Yaskawa INFORM job: DEMO_ROOF_UPPER_0625_3PAINT_43.JBI

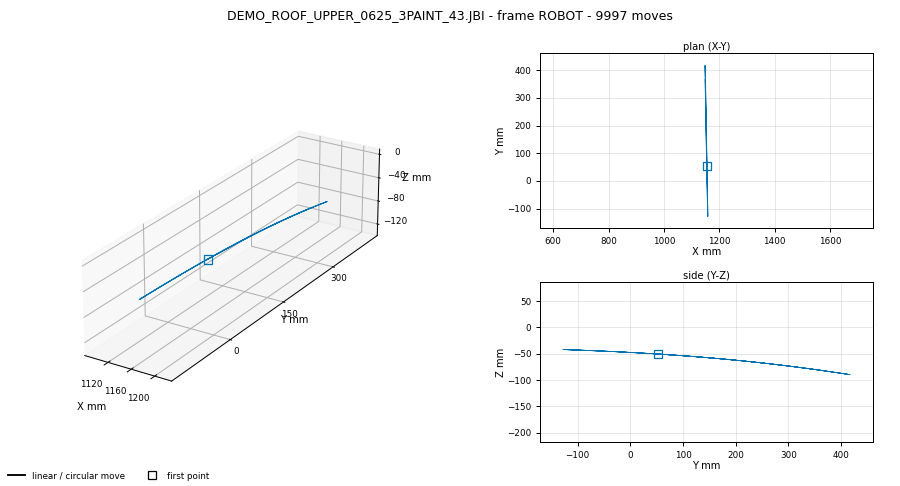
[picture p0: tool path of DEMO_ROOF_UPPER_0625_3PAINT_43.JBI in frame ROBOT, 9997 of 9997 moves have a stored position in this frame; points joined in program order, loops and branches not executed]
/JOB
//NAME DEMO_ROOF_UPPER_0625_3PAINT43
//POS
///NPOS 9997,0,0,0,0,0
///TOOL 0
///USER 0
///POSTYPE ROBOT
///RECTAN
///RCONF 1,0,0,0,0,0,0,0,0,0,0,0,0,0,0,0,0,0,0,0,0,0,0,0
C00000=1156.150,53.320,-50.344,-179.654,6.262,149.031
C00001=1156.144,53.589,-50.362,-179.651,6.263,149.031
C00002=1156.139,53.857,-50.379,-179.648,6.265,149.030
C00003=1156.133,54.126,-50.396,-179.646,6.265,149.030
C00004=1156.128,54.395,-50.413,-179.642,6.267,149.029
C00005=1156.123,54.644,-50.429,-179.640,6.268,149.028
C00006=1156.118,54.893,-50.445,-179.637,6.269,149.028
C00007=1156.113,55.143,-50.461,-179.635,6.270,149.027
C00008=1156.108,55.392,-50.476,-179.632,6.271,149.027
C00009=1156.103,55.641,-50.492,-179.629,6.272,149.026
C00010=1156.098,55.891,-50.508,-179.627,6.274,149.026
C00011=1156.093,56.141,-50.524,-179.624,6.274,149.025
C00012=1156.089,56.390,-50.540,-179.622,6.275,149.025
C00013=1156.083,56.639,-50.556,-179.619,6.277,149.024
C00014=1156.078,56.888,-50.572,-179.617,6.277,149.024
C00015=1156.073,57.138,-50.588,-179.614,6.279,149.023
C00016=1156.068,57.388,-50.604,-179.611,6.279,149.022
C00017=1156.063,57.637,-50.620,-179.608,6.281,149.022
C00018=1156.058,57.887,-50.636,-179.606,6.282,149.022
C00019=1156.054,58.136,-50.653,-179.603,6.283,149.021
C00020=1156.048,58.385,-50.668,-179.601,6.284,149.020
C00021=1156.044,58.635,-50.685,-179.598,6.285,149.020
C00022=1156.038,58.884,-50.700,-179.595,6.286,149.019
C00023=1156.033,59.133,-50.717,-179.592,6.287,149.019
C00024=1156.028,59.383,-50.733,-179.590,6.288,149.018
C00025=1156.023,59.632,-50.749,-179.587,6.290,149.018
C00026=1156.019,59.882,-50.765,-179.585,6.290,149.017
C00027=1156.013,60.131,-50.781,-179.582,6.292,149.017
C00028=1156.009,60.381,-50.797,-179.579,6.293,149.016
C00029=1156.004,60.630,-50.814,-179.577,6.294,149.016
C00030=1155.998,60.880,-50.830,-179.574,6.295,149.015
C00031=1155.993,61.129,-50.846,-179.571,6.296,149.015
C00032=1155.988,61.379,-50.862,-179.569,6.297,149.014
C00033=1155.983,61.628,-50.879,-179.566,6.298,149.013
C00034=1155.979,61.877,-50.895,-179.564,6.299,149.013
C00035=1155.973,62.127,-50.911,-179.561,6.301,149.013
C00036=1155.969,62.376,-50.928,-179.558,6.302,149.012
C00037=1155.963,62.626,-50.943,-179.556,6.303,149.011
C00038=1155.959,62.875,-50.960,-179.553,6.304,149.011
C00039=1155.954,63.124,-50.976,-179.550,6.305,149.010
C00040=1155.948,63.374,-50.993,-179.548,6.306,149.010
C00041=1155.944,63.624,-51.009,-179.545,6.307,149.009
C00042=1155.939,63.873,-51.026,-179.543,6.308,149.009
C00043=1155.934,64.123,-51.042,-179.539,6.310,149.008
C00044=1155.929,64.371,-51.058,-179.537,6.311,149.008
C00045=1155.924,64.621,-51.075,-179.535,6.312,149.007
C00046=1155.919,64.870,-51.092,-179.532,6.313,149.007
C00047=1155.914,65.120,-51.107,-179.529,6.314,149.006
C00048=1155.909,65.369,-51.124,-179.527,6.315,149.006
C00049=1155.904,65.618,-51.140,-179.524,6.317,149.005
C00050=1155.899,65.869,-51.156,-179.521,6.318,149.005
C00051=1155.894,66.118,-51.173,-179.518,6.319,149.004
C00052=1155.889,66.367,-51.190,-179.516,6.320,149.004
C00053=1155.884,66.616,-51.206,-179.514,6.321,149.003
C00054=1155.880,66.865,-51.223,-179.510,6.323,149.003
C00055=1155.875,67.115,-51.239,-179.508,6.323,149.002
C00056=1155.869,67.365,-51.256,-179.505,6.325,149.001
C00057=1155.864,67.614,-51.272,-179.503,6.326,149.001
C00058=1155.859,67.863,-51.289,-179.500,6.327,149.001
C00059=1155.855,68.112,-51.305,-179.497,6.328,149.000
C00060=1155.850,68.362,-51.323,-179.495,6.329,148.999
C00061=1155.844,68.612,-51.338,-179.492,6.330,148.999
C00062=1155.840,68.861,-51.355,-179.489,6.332,148.998
C00063=1155.835,69.111,-51.372,-179.487,6.333,148.998
C00064=1155.830,69.360,-51.389,-179.484,6.334,148.997
C00065=1155.825,69.609,-51.405,-179.481,6.335,148.997
C00066=1155.821,69.859,-51.422,-179.479,6.336,148.996
C00067=1155.815,70.108,-51.439,-179.476,6.338,148.996
C00068=1155.810,70.357,-51.455,-179.474,6.338,148.995
C00069=1155.806,70.607,-51.472,-179.470,6.340,148.995
C00070=1155.800,70.856,-51.489,-179.468,6.341,148.994
C00071=1155.796,71.105,-51.506,-179.466,6.342,148.994
C00072=1155.790,71.356,-51.522,-179.462,6.344,148.993
C00073=1155.785,71.604,-51.539,-179.460,6.344,148.993
C00074=1155.780,71.854,-51.555,-179.457,6.346,148.992
C00075=1155.775,72.104,-51.572,-179.455,6.347,148.992
C00076=1155.770,72.352,-51.589,-179.452,6.348,148.991
C00077=1155.766,72.602,-51.605,-179.449,6.350,148.991
C00078=1155.761,72.851,-51.623,-179.447,6.350,148.990
C00079=1155.756,73.100,-51.640,-179.444,6.352,148.990
C00080=1155.750,73.350,-51.657,-179.441,6.353,148.989
C00081=1155.746,73.599,-51.674,-179.439,6.354,148.989
C00082=1155.741,73.849,-51.690,-179.436,6.355,148.988
C00083=1155.736,74.098,-51.707,-179.433,6.357,148.987
C00084=1155.731,74.347,-51.724,-179.430,6.358,148.987
C00085=1155.726,74.597,-51.741,-179.428,6.359,148.987
C00086=1155.721,74.847,-51.758,-179.425,6.360,148.986
C00087=1155.716,75.096,-51.775,-179.423,6.361,148.986
C00088=1155.711,75.345,-51.791,-179.420,6.363,148.985
C00089=1155.706,75.595,-51.809,-179.417,6.364,148.984
C00090=1155.702,75.844,-51.826,-179.415,6.365,148.984
C00091=1155.696,76.093,-51.843,-179.412,6.367,148.984
C00092=1155.691,76.342,-51.860,-179.409,6.367,148.983
C00093=1155.686,76.592,-51.877,-179.407,6.369,148.983
C00094=1155.682,76.842,-51.894,-179.404,6.371,148.982
C00095=1155.676,77.091,-51.910,-179.401,6.371,148.981
C00096=1155.672,77.340,-51.928,-179.399,6.373,148.981
C00097=1155.667,77.589,-51.945,-179.396,6.373,148.980
C00098=1155.662,77.839,-51.962,-179.393,6.375,148.980
C00099=1155.657,78.089,-51.979,-179.391,6.377,148.979
C00100=1155.652,78.337,-51.996,-179.388,6.377,148.979
C00101=1155.647,78.587,-52.013,-179.385,6.379,148.978
C00102=1155.642,78.836,-52.030,-179.382,6.381,148.978
C00103=1155.637,79.086,-52.047,-179.380,6.381,148.977
C00104=1155.632,79.335,-52.065,-179.377,6.383,148.977
C00105=1155.627,79.603,-52.083,-179.374,6.384,148.976
C00106=1155.622,79.872,-52.102,-179.372,6.385,148.976
C00107=1155.616,80.141,-52.120,-179.369,6.387,148.975
C00108=1155.611,80.409,-52.138,-179.366,6.388,148.975
C00109=1155.606,80.658,-52.156,-179.363,6.390,148.974
C00110=1155.602,80.907,-52.173,-179.360,6.390,148.974
C00111=1155.596,81.157,-52.190,-179.358,6.392,148.973
C00112=1155.591,81.406,-52.208,-179.355,6.393,148.973
C00113=1155.586,81.655,-52.224,-179.352,6.394,148.972
C00114=1155.581,81.904,-52.242,-179.350,6.396,148.972
C00115=1155.576,82.154,-52.259,-179.347,6.397,148.971
C00116=1155.572,82.403,-52.276,-179.344,6.398,148.971
C00117=1155.567,82.653,-52.294,-179.341,6.400,148.970
C00118=1155.562,82.902,-52.311,-179.339,6.401,148.970
C00119=1155.557,83.151,-52.329,-179.336,6.402,148.969
C00120=1155.552,83.401,-52.346,-179.333,6.403,148.969
C00121=1155.547,83.650,-52.364,-179.331,6.404,148.968
C00122=1155.542,83.899,-52.380,-179.329,6.406,148.968
C00123=1155.537,84.148,-52.398,-179.325,6.407,148.967
C00124=1155.532,84.398,-52.416,-179.323,6.408,148.967
C00125=1155.527,84.647,-52.434,-179.320,6.410,148.966
C00126=1155.523,84.897,-52.450,-179.317,6.411,148.966
C00127=1155.518,85.146,-52.468,-179.315,6.412,148.965
C00128=1155.513,85.396,-52.485,-179.312,6.414,148.965
C00129=1155.508,85.645,-52.503,-179.309,6.415,148.964
C00130=1155.503,85.894,-52.520,-179.307,6.416,148.964
C00131=1155.498,86.143,-52.538,-179.304,6.418,148.963
C00132=1155.493,86.393,-52.555,-179.301,6.419,148.963
C00133=1155.488,86.642,-52.573,-179.299,6.420,148.962
C00134=1155.484,86.892,-52.590,-179.296,6.421,148.962
C00135=1155.479,87.141,-52.608,-179.293,6.423,148.961
C00136=1155.474,87.390,-52.626,-179.290,6.424,148.961
C00137=1155.469,87.640,-52.643,-179.288,6.425,148.960
C00138=1155.464,87.889,-52.661,-179.285,6.427,148.960
C00139=1155.460,88.138,-52.679,-179.282,6.428,148.959
C00140=1155.454,88.388,-52.696,-179.280,6.429,148.959
C00141=1155.449,88.637,-52.714,-179.277,6.431,148.959
C00142=1155.445,88.886,-52.732,-179.274,6.432,148.958
C00143=1155.439,89.136,-52.749,-179.272,6.433,148.957
C00144=1155.434,89.385,-52.767,-179.269,6.435,148.957
C00145=1155.429,89.634,-52.785,-179.266,6.437,148.957
C00146=1155.425,89.884,-52.802,-179.264,6.437,148.956
C00147=1155.420,90.133,-52.820,-179.261,6.439,148.956
C00148=1155.415,90.382,-52.838,-179.258,6.440,148.955
C00149=1155.410,90.631,-52.856,-179.255,6.442,148.954
C00150=1155.405,90.881,-52.873,-179.253,6.443,148.954
C00151=1155.400,91.130,-52.891,-179.250,6.444,148.954
C00152=1155.395,91.380,-52.909,-179.247,6.446,148.953
C00153=1155.390,91.629,-52.927,-179.245,6.446,148.953
C00154=1155.385,91.878,-52.944,-179.242,6.448,148.952
C00155=1155.380,92.128,-52.962,-179.239,6.450,148.952
C00156=1155.376,92.377,-52.979,-179.236,6.451,148.951
C00157=1155.371,92.626,-52.997,-179.234,6.452,148.951
C00158=1155.366,92.875,-53.015,-179.231,6.454,148.950
C00159=1155.361,93.124,-53.033,-179.229,6.455,148.950
C00160=1155.356,93.374,-53.051,-179.226,6.456,148.949
C00161=1155.351,93.623,-53.069,-179.223,6.458,148.949
C00162=1155.346,93.872,-53.087,-179.221,6.459,148.948
C00163=1155.342,94.122,-53.105,-179.218,6.461,148.948
C00164=1155.337,94.371,-53.123,-179.215,6.462,148.947
C00165=1155.332,94.620,-53.141,-179.212,6.463,148.947
C00166=1155.327,94.870,-53.159,-179.210,6.465,148.946
C00167=1155.322,95.119,-53.177,-179.207,6.466,148.946
C00168=1155.317,95.368,-53.195,-179.204,6.467,148.945
C00169=1155.312,95.617,-53.213,-179.202,6.469,148.945
C00170=1155.308,95.866,-53.231,-179.199,6.471,148.945
C00171=1155.303,96.115,-53.249,-179.196,6.471,148.944
C00172=1155.298,96.366,-53.268,-179.194,6.473,148.943
C00173=1155.292,96.615,-53.285,-179.191,6.474,148.943
C00174=1155.287,96.865,-53.303,-179.188,6.476,148.943
C00175=1155.283,97.113,-53.322,-179.185,6.477,148.942
C00176=1155.278,97.362,-53.340,-179.183,6.478,148.942
C00177=1155.273,97.612,-53.358,-179.180,6.480,148.941
C00178=1155.269,97.861,-53.376,-179.177,6.482,148.941
C00179=1155.264,98.111,-53.394,-179.174,6.483,148.940
C00180=1155.259,98.360,-53.412,-179.172,6.484,148.940
C00181=1155.254,98.609,-53.430,-179.169,6.486,148.939
C00182=1155.249,98.858,-53.448,-179.166,6.487,148.939
C00183=1155.243,99.108,-53.467,-179.163,6.489,148.938
C00184=1155.239,99.357,-53.485,-179.161,6.490,148.938
C00185=1155.234,99.607,-53.503,-179.158,6.491,148.937
C00186=1155.229,99.856,-53.521,-179.156,6.493,148.937
C00187=1155.224,100.105,-53.539,-179.152,6.494,148.936
C00188=1155.220,100.354,-53.557,-179.150,6.495,148.936
C00189=1155.215,100.604,-53.576,-179.148,6.497,148.935
C00190=1155.210,100.853,-53.594,-179.145,6.499,148.935
C00191=1155.205,101.102,-53.612,-179.142,6.500,148.934
C00192=1155.200,101.351,-53.630,-179.139,6.502,148.934
C00193=1155.196,101.601,-53.649,-179.137,6.502,148.934
C00194=1155.190,101.850,-53.668,-179.134,6.504,148.933
C00195=1155.185,102.099,-53.686,-179.131,6.506,148.933
C00196=1155.181,102.348,-53.704,-179.128,6.507,148.932
C00197=1155.176,102.598,-53.722,-179.126,6.508,148.932
C00198=1155.172,102.847,-53.741,-179.123,6.510,148.931
C00199=1155.166,103.096,-53.760,-179.121,6.511,148.931
C00200=1155.161,103.345,-53.778,-179.117,6.513,148.930
C00201=1155.157,103.595,-53.796,-179.115,6.514,148.930
C00202=1155.151,103.844,-53.815,-179.113,6.515,148.929
C00203=1155.146,104.093,-53.833,-179.110,6.517,148.929
C00204=1155.142,104.343,-53.851,-179.107,6.518,148.928
C00205=1155.138,104.592,-53.870,-179.104,6.520,148.928
C00206=1155.132,104.841,-53.889,-179.101,6.522,148.928
C00207=1155.127,105.090,-53.907,-179.099,6.523,148.927
C00208=1155.123,105.340,-53.926,-179.096,6.524,148.927
C00209=1155.117,105.608,-53.946,-179.093,6.526,148.926
C00210=1155.112,105.877,-53.965,-179.090,6.527,148.926
C00211=1155.107,106.145,-53.986,-179.087,6.529,148.925
C00212=1155.102,106.413,-54.006,-179.084,6.530,148.925
C00213=1155.096,106.663,-54.024,-179.082,6.532,148.924
C00214=1155.092,106.912,-54.043,-179.079,6.534,148.924
C00215=1155.088,107.161,-54.061,-179.076,6.536,148.923
C00216=1155.082,107.410,-54.081,-179.073,6.537,148.923
C00217=1155.077,107.659,-54.099,-179.070,6.539,148.922
C00218=1155.073,107.909,-54.118,-179.068,6.539,148.922
C00219=1155.068,108.158,-54.136,-179.065,6.541,148.922
C00220=1155.063,108.407,-54.155,-179.063,6.543,148.921
C00221=1155.058,108.657,-54.174,-179.060,6.544,148.921
C00222=1155.053,108.905,-54.193,-179.057,6.546,148.920
C00223=1155.048,109.155,-54.211,-179.054,6.548,148.920
C00224=1155.044,109.404,-54.230,-179.052,6.548,148.919
C00225=1155.039,109.653,-54.248,-179.049,6.550,148.919
C00226=1155.034,109.903,-54.268,-179.046,6.552,148.918
C00227=1155.029,110.152,-54.286,-179.043,6.553,148.918
C00228=1155.024,110.401,-54.305,-179.041,6.555,148.917
C00229=1155.019,110.651,-54.323,-179.038,6.557,148.917
C00230=1155.014,110.900,-54.343,-179.036,6.558,148.917
C00231=1155.010,111.149,-54.362,-179.033,6.559,148.916
C00232=1155.004,111.398,-54.380,-179.030,6.561,148.916
C00233=1155.000,111.647,-54.399,-179.027,6.562,148.915
C00234=1154.995,111.897,-54.418,-179.024,6.564,148.915
C00235=1154.990,112.146,-54.437,-179.022,6.566,148.914
C00236=1154.985,112.395,-54.456,-179.019,6.567,148.914
C00237=1154.981,112.645,-54.474,-179.016,6.568,148.913
C00238=1154.976,112.894,-54.494,-179.014,6.570,148.913
C00239=1154.971,113.143,-54.513,-179.011,6.571,148.913
C00240=1154.966,113.392,-54.531,-179.008,6.573,148.912
C00241=1154.961,113.642,-54.551,-179.005,6.575,148.912
C00242=1154.956,113.890,-54.570,-179.003,6.576,148.911
C00243=1154.951,114.140,-54.589,-178.999,6.578,148.911
C00244=1154.947,114.389,-54.607,-178.997,6.579,148.910
C00245=1154.942,114.639,-54.627,-178.995,6.580,148.910
C00246=1154.937,114.887,-54.646,-178.992,6.582,148.909
C00247=1154.932,115.137,-54.665,-178.989,6.584,148.909
C00248=1154.927,115.386,-54.684,-178.986,6.585,148.909
C00249=1154.923,115.635,-54.703,-178.983,6.587,148.908
C00250=1154.917,115.884,-54.722,-178.981,6.589,148.908
C00251=1154.913,116.134,-54.742,-178.978,6.590,148.907
C00252=1154.908,116.382,-54.761,-178.975,6.592,148.907
C00253=1154.903,116.632,-54.780,-178.973,6.593,148.906
C00254=1154.898,116.881,-54.798,-178.970,6.595,148.906
C00255=1154.894,117.131,-54.818,-178.968,6.596,148.906
C00256=1154.888,117.380,-54.837,-178.964,6.598,148.905
C00257=1154.884,117.629,-54.857,-178.962,6.599,148.905
C00258=1154.879,117.878,-54.876,-178.959,6.601,148.904
C00259=1154.874,118.127,-54.895,-178.956,6.603,148.904
C00260=1154.870,118.377,-54.915,-178.953,6.604,148.903
C00261=1154.865,118.625,-54.934,-178.951,6.606,148.903
C00262=1154.860,118.875,-54.953,-178.948,6.608,148.903
C00263=1154.855,119.124,-54.972,-178.945,6.608,148.902
C00264=1154.851,119.373,-54.992,-178.943,6.610,148.901
C00265=1154.845,119.623,-55.010,-178.940,6.612,148.901
C00266=1154.840,119.872,-55.030,-178.937,6.613,148.901
C00267=1154.836,120.122,-55.049,-178.935,6.615,148.900
C00268=1154.831,120.370,-55.068,-178.932,6.617,148.900
C00269=1154.826,120.620,-55.088,-178.929,6.619,148.899
C00270=1154.821,120.869,-55.107,-178.926,6.620,148.899
C00271=1154.817,121.118,-55.127,-178.923,6.622,148.898
C00272=1154.812,121.367,-55.147,-178.920,6.623,148.898
C00273=1154.807,121.616,-55.166,-178.918,6.625,148.898
C00274=1154.802,121.865,-55.185,-178.915,6.627,148.897
C00275=1154.797,122.114,-55.205,-178.912,6.629,148.897
C00276=1154.792,122.364,-55.224,-178.910,6.630,148.896
C00277=1154.788,122.613,-55.244,-178.907,6.631,148.896
C00278=1154.783,122.862,-55.263,-178.905,6.633,148.896
C00279=1154.778,123.112,-55.282,-178.902,6.634,148.895
C00280=1154.774,123.361,-55.302,-178.899,6.636,148.895
C00281=1154.768,123.610,-55.321,-178.896,6.638,148.894
C00282=1154.764,123.859,-55.342,-178.893,6.639,148.894
C00283=1154.759,124.108,-55.361,-178.891,6.641,148.893
C00284=1154.754,124.357,-55.380,-178.888,6.643,148.893
C00285=1154.750,124.607,-55.400,-178.885,6.644,148.893
C00286=1154.745,124.856,-55.419,-178.883,6.646,148.892
C00287=1154.740,125.104,-55.439,-178.880,6.648,148.892
C00288=1154.735,125.354,-55.459,-178.877,6.650,148.891
C00289=1154.730,125.604,-55.479,-178.874,6.651,148.891
C00290=1154.725,125.852,-55.498,-178.871,6.653,148.890
C00291=1154.721,126.101,-55.518,-178.868,6.654,148.890
C00292=1154.716,126.351,-55.538,-178.866,6.656,148.890
C00293=1154.711,126.600,-55.557,-178.863,6.658,148.889
C00294=1154.706,126.849,-55.577,-178.860,6.659,148.889
C00295=1154.701,127.098,-55.597,-178.858,6.661,148.888
C00296=1154.697,127.348,-55.616,-178.855,6.663,148.888
C00297=1154.692,127.596,-55.636,-178.852,6.665,148.888
C00298=1154.688,127.845,-55.656,-178.849,6.666,148.887
C00299=1154.683,128.095,-55.676,-178.847,6.667,148.887
C00300=1154.678,128.345,-55.695,-178.844,6.669,148.886
C00301=1154.673,128.593,-55.715,-178.841,6.670,148.886
C00302=1154.668,128.842,-55.735,-178.839,6.672,148.885
C00303=1154.664,129.092,-55.755,-178.836,6.674,148.885
C00304=1154.659,129.341,-55.775,-178.833,6.675,148.885
C00305=1154.654,129.590,-55.794,-178.831,6.677,148.884
C00306=1154.649,129.839,-55.815,-178.828,6.679,148.884
C00307=1154.644,130.089,-55.835,-178.825,6.681,148.883
C00308=1154.639,130.338,-55.855,-178.822,6.682,148.883
C00309=1154.634,130.586,-55.875,-178.820,6.684,148.883
C00310=1154.629,130.836,-55.894,-178.817,6.686,148.882
C00311=1154.625,131.085,-55.915,-178.814,6.687,148.882
C00312=1154.620,131.334,-55.934,-178.812,6.689,148.881
C00313=1154.616,131.602,-55.956,-178.808,6.691,148.881
C00314=1154.610,131.871,-55.978,-178.805,6.693,148.880
C00315=1154.605,132.140,-55.999,-178.802,6.695,148.880
C00316=1154.600,132.408,-56.021,-178.800,6.696,148.880
C00317=1154.595,132.658,-56.041,-178.797,6.698,148.879
C00318=1154.590,132.906,-56.061,-178.794,6.700,148.879
C00319=1154.585,133.156,-56.081,-178.792,6.702,148.879
C00320=1154.581,133.405,-56.101,-178.789,6.703,148.878
C00321=1154.576,133.654,-56.121,-178.786,6.705,148.878
C00322=1154.571,133.904,-56.142,-178.783,6.706,148.877
C00323=1154.566,134.153,-56.162,-178.780,6.708,148.877
C00324=1154.561,134.401,-56.181,-178.778,6.710,148.876
C00325=1154.557,134.650,-56.202,-178.775,6.712,148.876
C00326=1154.552,134.899,-56.222,-178.772,6.714,148.876
C00327=1154.547,135.149,-56.242,-178.769,6.716,148.875
C00328=1154.542,135.398,-56.263,-178.766,6.718,148.875
C00329=1154.538,135.647,-56.283,-178.763,6.719,148.874
C00330=1154.533,135.897,-56.303,-178.761,6.721,148.874
C00331=1154.529,136.146,-56.323,-178.758,6.723,148.874
C00332=1154.523,136.395,-56.344,-178.755,6.724,148.873
C00333=1154.518,136.644,-56.363,-178.753,6.726,148.873
C00334=1154.514,136.893,-56.384,-178.750,6.728,148.872
C00335=1154.509,137.142,-56.404,-178.747,6.730,148.872
C00336=1154.504,137.391,-56.425,-178.744,6.731,148.872
C00337=1154.499,137.640,-56.445,-178.742,6.733,148.871
C00338=1154.495,137.889,-56.465,-178.739,6.735,148.871
C00339=1154.490,138.139,-56.486,-178.736,6.736,148.870
C00340=1154.485,138.388,-56.506,-178.734,6.738,148.870
C00341=1154.481,138.637,-56.527,-178.731,6.740,148.870
C00342=1154.476,138.886,-56.546,-178.728,6.742,148.869
C00343=1154.471,139.135,-56.567,-178.725,6.743,148.869
C00344=1154.466,139.384,-56.588,-178.723,6.745,148.869
C00345=1154.462,139.633,-56.608,-178.720,6.747,148.868
C00346=1154.457,139.883,-56.629,-178.717,6.748,148.868
C00347=1154.452,140.132,-56.649,-178.714,6.751,148.867
C00348=1154.448,140.380,-56.670,-178.711,6.753,148.867
C00349=1154.442,140.630,-56.690,-178.709,6.754,148.867
C00350=1154.438,140.879,-56.710,-178.706,6.756,148.866
C00351=1154.433,141.129,-56.731,-178.703,6.758,148.866
C00352=1154.428,141.377,-56.752,-178.700,6.760,148.865
C00353=1154.424,141.626,-56.772,-178.698,6.761,148.865
C00354=1154.419,141.876,-56.793,-178.695,6.763,148.865
C00355=1154.414,142.125,-56.813,-178.692,6.765,148.864
C00356=1154.409,142.374,-56.834,-178.690,6.767,148.864
C00357=1154.405,142.623,-56.855,-178.687,6.768,148.864
C00358=1154.400,142.872,-56.875,-178.684,6.770,148.863
C00359=1154.395,143.121,-56.896,-178.682,6.772,148.863
C00360=1154.391,143.370,-56.917,-178.678,6.774,148.862
C00361=1154.386,143.619,-56.938,-178.676,6.776,148.862
C00362=1154.381,143.868,-56.958,-178.673,6.778,148.862
C00363=1154.376,144.117,-56.979,-178.670,6.779,148.861
C00364=1154.371,144.366,-56.999,-178.667,6.781,148.861
C00365=1154.366,144.616,-57.020,-178.665,6.783,148.860
C00366=1154.362,144.864,-57.041,-178.662,6.785,148.860
C00367=1154.357,145.113,-57.062,-178.659,6.786,148.860
C00368=1154.353,145.362,-57.083,-178.657,6.788,148.859
C00369=1154.347,145.611,-57.104,-178.654,6.790,148.859
C00370=1154.343,145.860,-57.124,-178.651,6.792,148.859
C00371=1154.338,146.110,-57.145,-178.648,6.794,148.858
C00372=1154.334,146.359,-57.166,-178.645,6.796,148.858
C00373=1154.329,146.608,-57.187,-178.643,6.798,148.858
C00374=1154.325,146.857,-57.208,-178.640,6.800,148.857
C00375=1154.319,147.106,-57.229,-178.638,6.801,148.857
C00376=1154.315,147.355,-57.249,-178.635,6.803,148.856
C00377=1154.310,147.604,-57.270,-178.632,6.805,148.856
C00378=1154.305,147.853,-57.292,-178.629,6.806,148.856
C00379=1154.301,148.102,-57.312,-178.626,6.809,148.855
C00380=1154.296,148.352,-57.333,-178.623,6.811,148.855
C00381=1154.292,148.601,-57.354,-178.621,6.812,148.855
C00382=1154.287,148.850,-57.375,-178.618,6.814,148.854
C00383=1154.281,149.099,-57.396,-178.615,6.816,148.854
C00384=1154.277,149.348,-57.417,-178.613,6.818,148.853
C00385=1154.272,149.597,-57.438,-178.610,6.819,148.853
C00386=1154.267,149.846,-57.459,-178.607,6.822,148.853
C00387=1154.263,150.095,-57.480,-178.604,6.824,148.852
C00388=1154.258,150.345,-57.501,-178.601,6.825,148.852
C00389=1154.253,150.593,-57.523,-178.598,6.827,148.851
C00390=1154.249,150.842,-57.543,-178.596,6.829,148.851
C00391=1154.244,151.091,-57.565,-178.594,6.831,148.851
C00392=1154.239,151.341,-57.586,-178.591,6.833,148.851
C00393=1154.235,151.590,-57.607,-178.588,6.835,148.850
C00394=1154.230,151.838,-57.628,-178.585,6.837,148.850
C00395=1154.225,152.088,-57.649,-178.582,6.839,148.849
C00396=1154.220,152.336,-57.671,-178.579,6.840,148.849
C00397=1154.216,152.586,-57.692,-178.577,6.842,148.849
C00398=1154.211,152.835,-57.713,-178.574,6.844,148.848
C00399=1154.206,153.084,-57.734,-178.571,6.846,148.848
C00400=1154.201,153.333,-57.755,-178.568,6.848,148.848
C00401=1154.197,153.581,-57.776,-178.566,6.850,148.847
C00402=1154.192,153.831,-57.798,-178.563,6.852,148.847
C00403=1154.187,154.080,-57.819,-178.560,6.854,148.847
C00404=1154.182,154.329,-57.840,-178.558,6.855,148.846
C00405=1154.177,154.578,-57.862,-178.554,6.858,148.846
C00406=1154.174,154.827,-57.883,-178.552,6.860,148.846
C00407=1154.168,155.076,-57.904,-178.549,6.861,148.845
C00408=1154.164,155.325,-57.926,-178.546,6.863,148.845
C00409=1154.159,155.575,-57.947,-178.544,6.865,148.844
C00410=1154.154,155.823,-57.969,-178.541,6.867,148.844
C00411=1154.149,156.073,-57.990,-178.538,6.869,148.844
C00412=1154.145,156.321,-58.011,-178.535,6.871,148.843
C00413=1154.141,156.570,-58.033,-178.533,6.873,148.843
C00414=1154.135,156.820,-58.054,-178.530,6.875,148.843
C00415=1154.131,157.068,-58.076,-178.527,6.876,148.842
C00416=1154.126,157.318,-58.098,-178.524,6.879,148.842
C00417=1154.122,157.587,-58.121,-178.521,6.881,148.842
C00418=1154.115,157.855,-58.144,-178.518,6.883,148.841
C00419=1154.111,158.124,-58.167,-178.515,6.885,148.841
C00420=1154.106,158.393,-58.191,-178.513,6.887,148.841
C00421=1154.101,158.642,-58.213,-178.509,6.889,148.840
C00422=1154.096,158.892,-58.234,-178.507,6.891,148.840
C00423=1154.091,159.140,-58.255,-178.504,6.893,148.839
C00424=1154.087,159.390,-58.277,-178.502,6.895,148.839
C00425=1154.082,159.638,-58.299,-178.499,6.896,148.839
C00426=1154.077,159.888,-58.320,-178.496,6.899,148.839
C00427=1154.073,160.137,-58.342,-178.493,6.901,148.838
C00428=1154.068,160.386,-58.364,-178.490,6.902,148.838
C00429=1154.064,160.635,-58.386,-178.488,6.904,148.837
C00430=1154.059,160.884,-58.407,-178.484,6.907,148.837
C00431=1154.053,161.133,-58.428,-178.482,6.909,148.837
C00432=1154.049,161.382,-58.450,-178.479,6.911,148.836
C00433=1154.044,161.631,-58.472,-178.477,6.912,148.836
C00434=1154.040,161.880,-58.494,-178.474,6.914,148.836
C00435=1154.035,162.129,-58.516,-178.471,6.917,148.835
C00436=1154.030,162.377,-58.538,-178.468,6.918,148.835
C00437=1154.026,162.627,-58.560,-178.466,6.920,148.835
C00438=1154.021,162.875,-58.581,-178.463,6.922,148.834
C00439=1154.017,163.125,-58.603,-178.460,6.925,148.834
C00440=1154.012,163.373,-58.625,-178.457,6.926,148.834
C00441=1154.008,163.623,-58.647,-178.454,6.928,148.833
C00442=1154.003,163.871,-58.669,-178.452,6.930,148.833
C00443=1153.998,164.120,-58.690,-178.449,6.933,148.833
C00444=1153.994,164.369,-58.712,-178.446,6.935,148.832
C00445=1153.989,164.618,-58.734,-178.444,6.936,148.832
C00446=1153.985,164.867,-58.756,-178.441,6.938,148.832
C00447=1153.979,165.116,-58.778,-178.438,6.941,148.831
C00448=1153.975,165.366,-58.800,-178.435,6.943,148.831
C00449=1153.970,165.614,-58.822,-178.433,6.944,148.831
C00450=1153.966,165.864,-58.844,-178.430,6.946,148.831
C00451=1153.961,166.112,-58.866,-178.427,6.949,148.830
C00452=1153.956,166.362,-58.888,-178.424,6.950,148.830
C00453=1153.952,166.610,-58.910,-178.421,6.952,148.829
C00454=1153.947,166.860,-58.932,-178.419,6.954,148.829
C00455=1153.942,167.108,-58.954,-178.416,6.957,148.829
C00456=1153.937,167.358,-58.976,-178.413,6.959,148.829
C00457=1153.933,167.606,-58.998,-178.410,6.960,148.828
C00458=1153.929,167.855,-59.020,-178.407,6.963,148.828
C00459=1153.923,168.104,-59.043,-178.405,6.965,148.828
C00460=1153.919,168.353,-59.065,-178.402,6.967,148.827
C00461=1153.914,168.602,-59.086,-178.399,6.968,148.827
C00462=1153.910,168.851,-59.109,-178.396,6.971,148.827
C00463=1153.905,169.100,-59.132,-178.394,6.973,148.826
C00464=1153.900,169.349,-59.154,-178.391,6.975,148.826
C00465=1153.896,169.598,-59.176,-178.388,6.977,148.826
C00466=1153.890,169.847,-59.198,-178.385,6.979,148.825
C00467=1153.886,170.096,-59.221,-178.383,6.981,148.825
C00468=1153.881,170.345,-59.242,-178.380,6.983,148.825
C00469=1153.877,170.594,-59.264,-178.377,6.985,148.824
C00470=1153.871,170.843,-59.287,-178.374,6.987,148.824
C00471=1153.868,171.092,-59.309,-178.372,6.989,148.824
C00472=1153.863,171.341,-59.331,-178.369,6.992,148.824
C00473=1153.858,171.590,-59.354,-178.366,6.994,148.823
C00474=1153.854,171.839,-59.376,-178.364,6.995,148.823
C00475=1153.849,172.087,-59.398,-178.360,6.998,148.823
C00476=1153.844,172.336,-59.422,-178.358,7.000,148.822
C00477=1153.840,172.586,-59.444,-178.355,7.002,148.822
C00478=1153.834,172.835,-59.466,-178.353,7.003,148.822
C00479=1153.830,173.083,-59.489,-178.349,7.006,148.821
C00480=1153.826,173.333,-59.511,-178.347,7.008,148.821
C00481=1153.821,173.581,-59.534,-178.344,7.010,148.821
C00482=1153.816,173.831,-59.556,-178.341,7.012,148.820
C00483=1153.811,174.080,-59.578,-178.338,7.014,148.820
C00484=1153.807,174.328,-59.601,-178.336,7.016,148.820
C00485=1153.803,174.578,-59.623,-178.333,7.019,148.820
C00486=1153.798,174.827,-59.646,-178.330,7.020,148.819
C00487=1153.793,175.075,-59.668,-178.328,7.022,148.819
C00488=1153.788,175.324,-59.691,-178.325,7.025,148.819
C00489=1153.784,175.574,-59.713,-178.322,7.027,148.818
C00490=1153.779,175.822,-59.736,-178.319,7.029,148.818
C00491=1153.775,176.071,-59.759,-178.316,7.031,148.818
C00492=1153.770,176.320,-59.782,-178.314,7.033,148.817
C00493=1153.765,176.568,-59.804,-178.311,7.035,148.817
C00494=1153.760,176.818,-59.827,-178.308,7.038,148.817
C00495=1153.756,177.067,-59.849,-178.305,7.039,148.816
C00496=1153.751,177.316,-59.872,-178.303,7.041,148.816
C00497=1153.747,177.564,-59.894,-178.300,7.044,148.816
C00498=1153.742,177.813,-59.918,-178.297,7.046,148.816
C00499=1153.738,178.063,-59.940,-178.295,7.048,148.815
C00500=1153.732,178.311,-59.963,-178.292,7.050,148.815
C00501=1153.728,178.560,-59.986,-178.289,7.052,148.815
C00502=1153.723,178.809,-60.008,-178.286,7.055,148.814
C00503=1153.720,179.058,-60.031,-178.283,7.057,148.814
C00504=1153.714,179.306,-60.054,-178.281,7.059,148.814
C00505=1153.710,179.555,-60.077,-178.277,7.061,148.814
C00506=1153.705,179.805,-60.099,-178.275,7.063,148.813
C00507=1153.701,180.054,-60.123,-178.272,7.065,148.813
C00508=1153.697,180.303,-60.146,-178.269,7.067,148.813
C00509=1153.691,180.551,-60.169,-178.267,7.070,148.813
C00510=1153.686,180.801,-60.191,-178.264,7.071,148.812
C00511=1153.682,181.049,-60.214,-178.261,7.074,148.812
C00512=1153.678,181.298,-60.237,-178.259,7.076,148.812
C00513=1153.672,181.547,-60.260,-178.256,7.079,148.811
C00514=1153.668,181.795,-60.283,-178.253,7.080,148.811
C00515=1153.663,182.045,-60.306,-178.251,7.082,148.811
C00516=1153.659,182.294,-60.329,-178.247,7.085,148.810
C00517=1153.655,182.543,-60.352,-178.245,7.087,148.810
C00518=1153.650,182.792,-60.375,-178.241,7.089,148.810
C00519=1153.645,183.040,-60.398,-178.239,7.091,148.810
C00520=1153.641,183.289,-60.421,-178.237,7.093,148.809
C00521=1153.635,183.559,-60.446,-178.233,7.096,148.809
C00522=1153.630,183.828,-60.471,-178.230,7.099,148.809
C00523=1153.626,184.099,-60.496,-178.228,7.100,148.808
C00524=1153.621,184.368,-60.521,-178.224,7.103,148.808
C00525=1153.615,184.617,-60.544,-178.222,7.105,148.808
C00526=1153.611,184.866,-60.567,-178.219,7.108,148.808
C00527=1153.607,185.114,-60.590,-178.216,7.109,148.807
C00528=1153.602,185.363,-60.613,-178.213,7.112,148.807
C00529=1153.597,185.612,-60.637,-178.211,7.114,148.807
C00530=1153.593,185.862,-60.660,-178.208,7.116,148.806
C00531=1153.588,186.111,-60.683,-178.205,7.118,148.806
C00532=1153.584,186.359,-60.707,-178.203,7.120,148.806
C00533=1153.580,186.608,-60.730,-178.199,7.123,148.806
C00534=1153.575,186.857,-60.754,-178.197,7.125,148.805
C00535=1153.570,187.105,-60.777,-178.194,7.128,148.805
C00536=1153.565,187.354,-60.800,-178.191,7.129,148.805
C00537=1153.560,187.603,-60.823,-178.189,7.131,148.805
C00538=1153.556,187.852,-60.846,-178.186,7.134,148.804
C00539=1153.552,188.101,-60.869,-178.183,7.136,148.804
C00540=1153.547,188.350,-60.893,-178.180,7.139,148.804
C00541=1153.542,188.599,-60.916,-178.178,7.140,148.804
C00542=1153.538,188.847,-60.940,-178.174,7.143,148.803
C00543=1153.533,189.096,-60.964,-178.172,7.145,148.803
C00544=1153.528,189.345,-60.987,-178.169,7.147,148.803
C00545=1153.524,189.594,-61.010,-178.167,7.150,148.803
C00546=1153.519,189.843,-61.034,-178.164,7.151,148.802
C00547=1153.515,190.092,-61.058,-178.161,7.154,148.802
C00548=1153.510,190.341,-61.081,-178.158,7.156,148.802
C00549=1153.505,190.590,-61.105,-178.155,7.159,148.801
C00550=1153.501,190.839,-61.128,-178.153,7.161,148.801
C00551=1153.497,191.087,-61.151,-178.150,7.163,148.801
C00552=1153.492,191.336,-61.175,-178.147,7.165,148.801
C00553=1153.487,191.585,-61.198,-178.145,7.167,148.800
C00554=1153.483,191.834,-61.222,-178.141,7.170,148.800
C00555=1153.478,192.083,-61.245,-178.139,7.172,148.800
C00556=1153.474,192.332,-61.269,-178.136,7.174,148.800
C00557=1153.469,192.580,-61.293,-178.133,7.176,148.799
C00558=1153.464,192.829,-61.317,-178.131,7.179,148.799
C00559=1153.459,193.078,-61.340,-178.128,7.181,148.799
C00560=1153.455,193.327,-61.364,-178.125,7.184,148.799
C00561=1153.450,193.576,-61.388,-178.122,7.186,148.798
C00562=1153.446,193.824,-61.412,-178.120,7.188,148.798
C00563=1153.441,194.073,-61.435,-178.117,7.190,148.798
C00564=1153.436,194.322,-61.458,-178.114,7.193,148.798
C00565=1153.432,194.571,-61.483,-178.111,7.195,148.797
C00566=1153.427,194.820,-61.506,-178.108,7.197,148.797
C00567=1153.423,195.068,-61.530,-178.106,7.200,148.797
C00568=1153.418,195.317,-61.553,-178.103,7.202,148.797
C00569=1153.414,195.566,-61.578,-178.100,7.204,148.797
C00570=1153.410,195.815,-61.601,-178.098,7.206,148.796
C00571=1153.404,196.064,-61.626,-178.095,7.209,148.796
C00572=1153.400,196.313,-61.649,-178.092,7.211,148.796
C00573=1153.395,196.562,-61.673,-178.089,7.213,148.795
C00574=1153.391,196.810,-61.697,-178.087,7.215,148.795
C00575=1153.386,197.059,-61.721,-178.084,7.218,148.795
C00576=1153.382,197.307,-61.745,-178.081,7.220,148.795
C00577=1153.377,197.557,-61.769,-178.078,7.223,148.794
C00578=1153.373,197.806,-61.793,-178.076,7.225,148.794
C00579=1153.368,198.054,-61.817,-178.073,7.227,148.794
C00580=1153.364,198.303,-61.841,-178.070,7.229,148.794
C00581=1153.359,198.552,-61.865,-178.067,7.232,148.794
C00582=1153.354,198.801,-61.889,-178.065,7.234,148.793
C00583=1153.349,199.049,-61.913,-178.062,7.237,148.793
C00584=1153.345,199.299,-61.937,-178.059,7.239,148.793
C00585=1153.341,199.547,-61.961,-178.056,7.241,148.793
C00586=1153.336,199.796,-61.985,-178.053,7.244,148.792
C00587=1153.331,200.045,-62.009,-178.051,7.246,148.792
C00588=1153.327,200.293,-62.033,-178.047,7.248,148.792
C00589=1153.323,200.543,-62.057,-178.045,7.251,148.792
C00590=1153.318,200.792,-62.082,-178.042,7.253,148.791
C00591=1153.313,201.040,-62.106,-178.040,7.255,148.791
C00592=1153.309,201.288,-62.130,-178.036,7.258,148.791
C00593=1153.304,201.537,-62.154,-178.034,7.260,148.791
C00594=1153.300,201.787,-62.178,-178.031,7.262,148.790
C00595=1153.295,202.035,-62.202,-178.029,7.265,148.790
C00596=1153.291,202.284,-62.226,-178.025,7.267,148.790
C00597=1153.286,202.532,-62.251,-178.023,7.269,148.790
C00598=1153.282,202.782,-62.275,-178.020,7.272,148.790
C00599=1153.278,203.030,-62.300,-178.018,7.274,148.789
C00600=1153.272,203.279,-62.324,-178.015,7.277,148.789
C00601=1153.268,203.528,-62.348,-178.012,7.279,148.789
C00602=1153.264,203.777,-62.372,-178.009,7.281,148.789
C00603=1153.259,204.026,-62.397,-178.006,7.284,148.789
C00604=1153.254,204.274,-62.421,-178.004,7.286,148.788
C00605=1153.249,204.523,-62.445,-178.001,7.289,148.788
C00606=1153.245,204.772,-62.470,-177.999,7.291,148.788
C00607=1153.240,205.021,-62.495,-177.995,7.293,148.788
C00608=1153.236,205.269,-62.519,-177.993,7.296,148.788
C00609=1153.232,205.518,-62.543,-177.990,7.298,148.787
C00610=1153.227,205.767,-62.568,-177.987,7.301,148.787
C00611=1153.223,206.015,-62.592,-177.984,7.303,148.787
C00612=1153.217,206.264,-62.616,-177.982,7.306,148.787
C00613=1153.214,206.513,-62.641,-177.979,7.308,148.786
C00614=1153.209,206.762,-62.666,-177.976,7.310,148.786
C00615=1153.204,207.010,-62.690,-177.973,7.312,148.786
C00616=1153.200,207.260,-62.715,-177.971,7.315,148.786
C00617=1153.195,207.508,-62.739,-177.968,7.318,148.786
C00618=1153.190,207.756,-62.764,-177.965,7.320,148.785
C00619=1153.187,208.005,-62.789,-177.962,7.323,148.785
C00620=1153.181,208.254,-62.813,-177.960,7.324,148.785
C00621=1153.178,208.503,-62.838,-177.957,7.327,148.785
C00622=1153.173,208.752,-62.862,-177.954,7.329,148.784
C00623=1153.167,209.001,-62.887,-177.951,7.332,148.784
C00624=1153.164,209.250,-62.911,-177.948,7.335,148.784
C00625=1153.158,209.520,-62.938,-177.945,7.338,148.784
C00626=1153.154,209.791,-62.965,-177.943,7.339,148.784
C00627=1153.149,210.061,-62.992,-177.940,7.342,148.783
C00628=1153.144,210.332,-63.019,-177.937,7.345,148.783
C00629=1153.139,210.580,-63.044,-177.934,7.348,148.783
C00630=1153.134,210.829,-63.069,-177.931,7.350,148.783
C00631=1153.130,211.078,-63.094,-177.928,7.352,148.783
C00632=1153.125,211.326,-63.118,-177.926,7.355,148.783
C00633=1153.121,211.575,-63.144,-177.923,7.357,148.782
C00634=1153.117,211.824,-63.168,-177.920,7.360,148.782
C00635=1153.112,212.072,-63.193,-177.917,7.363,148.782
C00636=1153.107,212.321,-63.218,-177.915,7.365,148.782
C00637=1153.103,212.570,-63.243,-177.912,7.368,148.782
C00638=1153.098,212.819,-63.268,-177.909,7.369,148.781
C00639=1153.094,213.067,-63.293,-177.906,7.372,148.781
C00640=1153.090,213.316,-63.317,-177.903,7.375,148.781
C00641=1153.085,213.564,-63.343,-177.901,7.377,148.781
C00642=1153.080,213.814,-63.368,-177.898,7.380,148.781
C00643=1153.076,214.062,-63.392,-177.896,7.382,148.780
C00644=1153.072,214.311,-63.418,-177.893,7.385,148.780
C00645=1153.067,214.560,-63.442,-177.889,7.387,148.780
C00646=1153.062,214.808,-63.468,-177.887,7.389,148.780
C00647=1153.058,215.057,-63.492,-177.884,7.392,148.780
C00648=1153.054,215.306,-63.518,-177.881,7.395,148.779
C00649=1153.049,215.554,-63.543,-177.879,7.397,148.779
C00650=1153.045,215.803,-63.568,-177.876,7.400,148.779
C00651=1153.039,216.052,-63.593,-177.873,7.402,148.779
C00652=1153.036,216.300,-63.618,-177.871,7.405,148.779
C00653=1153.031,216.549,-63.643,-177.868,7.407,148.779
C00654=1153.027,216.798,-63.669,-177.865,7.409,148.778
C00655=1153.021,217.047,-63.693,-177.862,7.412,148.778
C00656=1153.017,217.295,-63.719,-177.859,7.415,148.778
C00657=1153.013,217.543,-63.744,-177.857,7.417,148.778
C00658=1153.009,217.793,-63.769,-177.854,7.420,148.778
C00659=1153.004,218.041,-63.795,-177.851,7.422,148.777
C00660=1153.000,218.290,-63.820,-177.849,7.424,148.777
C00661=1152.995,218.539,-63.845,-177.846,7.427,148.777
C00662=1152.990,218.787,-63.870,-177.843,7.430,148.777
C00663=1152.986,219.036,-63.896,-177.841,7.432,148.777
C00664=1152.981,219.285,-63.921,-177.838,7.435,148.777
C00665=1152.977,219.533,-63.946,-177.834,7.438,148.776
C00666=1152.973,219.782,-63.972,-177.832,7.440,148.776
C00667=1152.968,220.031,-63.996,-177.830,7.443,148.776
C00668=1152.964,220.279,-64.022,-177.826,7.445,148.776
C00669=1152.959,220.528,-64.048,-177.824,7.447,148.776
C00670=1152.955,220.776,-64.073,-177.821,7.450,148.775
C00671=1152.950,221.025,-64.099,-177.818,7.453,148.775
C00672=1152.945,221.274,-64.124,-177.815,7.456,148.775
C00673=1152.941,221.523,-64.149,-177.813,7.458,148.775
C00674=1152.937,221.772,-64.175,-177.810,7.460,148.775
C00675=1152.932,222.020,-64.201,-177.807,7.463,148.775
C00676=1152.928,222.268,-64.226,-177.805,7.465,148.774
C00677=1152.924,222.517,-64.252,-177.802,7.468,148.774
C00678=1152.918,222.766,-64.277,-177.799,7.471,148.774
C00679=1152.914,223.015,-64.302,-177.797,7.473,148.774
C00680=1152.910,223.264,-64.328,-177.794,7.476,148.774
C00681=1152.905,223.512,-64.354,-177.790,7.479,148.774
C00682=1152.901,223.760,-64.379,-177.788,7.482,148.773
C00683=1152.897,224.009,-64.405,-177.785,7.484,148.773
C00684=1152.892,224.257,-64.431,-177.782,7.486,148.773
C00685=1152.888,224.506,-64.456,-177.779,7.489,148.773
C00686=1152.883,224.755,-64.483,-177.777,7.491,148.773
C00687=1152.878,225.003,-64.508,-177.774,7.494,148.773
C00688=1152.874,225.252,-64.534,-177.771,7.497,148.772
C00689=1152.869,225.501,-64.559,-177.768,7.500,148.772
C00690=1152.865,225.750,-64.585,-177.766,7.502,148.772
C00691=1152.860,225.998,-64.611,-177.763,7.505,148.772
C00692=1152.856,226.247,-64.636,-177.760,7.507,148.772
C00693=1152.852,226.496,-64.662,-177.758,7.509,148.772
C00694=1152.847,226.745,-64.688,-177.755,7.512,148.772
C00695=1152.842,226.993,-64.714,-177.752,7.515,148.771
C00696=1152.838,227.242,-64.740,-177.749,7.518,148.771
C00697=1152.834,227.490,-64.765,-177.747,7.520,148.771
C00698=1152.830,227.739,-64.792,-177.744,7.523,148.771
C00699=1152.825,227.987,-64.817,-177.741,7.526,148.771
C00700=1152.820,228.236,-64.844,-177.738,7.528,148.771
C00701=1152.816,228.485,-64.869,-177.736,7.531,148.771
C00702=1152.812,228.733,-64.895,-177.733,7.533,148.770
C00703=1152.807,228.981,-64.920,-177.730,7.536,148.770
C00704=1152.802,229.230,-64.948,-177.727,7.539,148.770
C00705=1152.798,229.479,-64.973,-177.725,7.541,148.770
C00706=1152.794,229.728,-64.999,-177.722,7.544,148.770
C00707=1152.789,229.976,-65.025,-177.719,7.547,148.770
C00708=1152.785,230.225,-65.052,-177.716,7.550,148.770
C00709=1152.780,230.473,-65.077,-177.714,7.552,148.769
C00710=1152.776,230.722,-65.103,-177.711,7.555,148.769
C00711=1152.771,230.971,-65.129,-177.708,7.558,148.769
C00712=1152.767,231.219,-65.156,-177.705,7.560,148.769
C00713=1152.763,231.468,-65.182,-177.703,7.562,148.769
C00714=1152.758,231.717,-65.208,-177.700,7.565,148.769
C00715=1152.753,231.964,-65.234,-177.697,7.568,148.769
C00716=1152.749,232.213,-65.260,-177.694,7.571,148.768
C00717=1152.744,232.462,-65.287,-177.692,7.573,148.768
C00718=1152.740,232.711,-65.313,-177.689,7.576,148.768
C00719=1152.736,232.959,-65.338,-177.686,7.579,148.768
C00720=1152.731,233.208,-65.365,-177.683,7.582,148.768
C00721=1152.727,233.457,-65.391,-177.680,7.584,148.768
C00722=1152.723,233.705,-65.418,-177.678,7.586,148.768
C00723=1152.717,233.953,-65.444,-177.675,7.589,148.768
C00724=1152.713,234.201,-65.470,-177.672,7.592,148.767
C00725=1152.709,234.451,-65.496,-177.670,7.595,148.767
C00726=1152.705,234.699,-65.523,-177.667,7.597,148.767
C00727=1152.700,234.948,-65.549,-177.664,7.600,148.767
C00728=1152.696,235.196,-65.576,-177.661,7.603,148.767
C00729=1152.690,235.468,-65.604,-177.659,7.606,148.767
C00730=1152.686,235.740,-65.633,-177.655,7.608,148.766
C00731=1152.680,236.012,-65.662,-177.652,7.612,148.766
C00732=1152.677,236.284,-65.691,-177.649,7.615,148.766
C00733=1152.672,236.532,-65.718,-177.647,7.617,148.766
C00734=1152.667,236.780,-65.743,-177.644,7.620,148.766
C00735=1152.663,237.029,-65.770,-177.641,7.623,148.766
C00736=1152.659,237.277,-65.797,-177.638,7.625,148.766
C00737=1152.654,237.526,-65.823,-177.635,7.628,148.766
C00738=1152.650,237.774,-65.850,-177.633,7.631,148.766
C00739=1152.645,238.023,-65.877,-177.631,7.633,148.766
C00740=1152.641,238.272,-65.902,-177.628,7.636,148.765
C00741=1152.636,238.520,-65.929,-177.624,7.639,148.765
C00742=1152.632,238.769,-65.956,-177.622,7.642,148.765
C00743=1152.627,239.017,-65.982,-177.619,7.645,148.765
C00744=1152.623,239.266,-66.009,-177.617,7.647,148.765
C00745=1152.619,239.514,-66.036,-177.614,7.650,148.765
C00746=1152.614,239.763,-66.063,-177.611,7.653,148.765
C00747=1152.609,240.012,-66.089,-177.608,7.656,148.765
C00748=1152.605,240.260,-66.116,-177.605,7.658,148.764
C00749=1152.601,240.508,-66.143,-177.602,7.661,148.764
C00750=1152.597,240.758,-66.170,-177.600,7.663,148.764
C00751=1152.593,241.006,-66.197,-177.597,7.666,148.764
C00752=1152.588,241.255,-66.223,-177.595,7.669,148.764
C00753=1152.584,241.503,-66.249,-177.592,7.672,148.764
C00754=1152.579,241.752,-66.276,-177.589,7.675,148.764
C00755=1152.574,242.000,-66.304,-177.586,7.678,148.764
C00756=1152.570,242.249,-66.331,-177.584,7.680,148.763
C00757=1152.566,242.497,-66.357,-177.581,7.683,148.763
C00758=1152.561,242.745,-66.384,-177.578,7.686,148.763
C00759=1152.557,242.994,-66.411,-177.575,7.689,148.763
C00760=1152.553,243.242,-66.438,-177.572,7.692,148.763
C00761=1152.548,243.490,-66.465,-177.570,7.695,148.763
C00762=1152.543,243.739,-66.492,-177.567,7.697,148.763
C00763=1152.539,243.988,-66.519,-177.565,7.700,148.763
C00764=1152.535,244.236,-66.546,-177.562,7.702,148.763
C00765=1152.531,244.485,-66.573,-177.559,7.705,148.763
C00766=1152.526,244.733,-66.600,-177.556,7.708,148.763
C00767=1152.521,244.982,-66.627,-177.553,7.711,148.762
C00768=1152.517,245.230,-66.653,-177.550,7.714,148.762
C00769=1152.513,245.479,-66.680,-177.548,7.717,148.762
C00770=1152.509,245.728,-66.708,-177.545,7.719,148.762
C00771=1152.504,245.976,-66.735,-177.543,7.722,148.762
C00772=1152.499,246.225,-66.762,-177.540,7.725,148.762
C00773=1152.495,246.473,-66.789,-177.537,7.728,148.762
C00774=1152.491,246.721,-66.815,-177.534,7.731,148.762
C00775=1152.486,246.970,-66.843,-177.531,7.734,148.762
C00776=1152.482,247.218,-66.871,-177.529,7.737,148.762
C00777=1152.478,247.467,-66.898,-177.526,7.739,148.762
C00778=1152.473,247.715,-66.925,-177.523,7.741,148.761
C00779=1152.468,247.964,-66.952,-177.520,7.744,148.761
C00780=1152.464,248.212,-66.979,-177.518,7.747,148.761
C00781=1152.460,248.461,-67.007,-177.515,7.750,148.761
C00782=1152.455,248.710,-67.034,-177.512,7.753,148.761
C00783=1152.451,248.958,-67.061,-177.509,7.756,148.761
C00784=1152.447,249.206,-67.088,-177.507,7.759,148.761
C00785=1152.442,249.454,-67.115,-177.504,7.762,148.761
C00786=1152.438,249.703,-67.143,-177.502,7.764,148.761
C00787=1152.434,249.952,-67.170,-177.499,7.767,148.761
C00788=1152.429,250.200,-67.198,-177.496,7.770,148.761
C00789=1152.425,250.448,-67.225,-177.493,7.773,148.761
C00790=1152.421,250.697,-67.252,-177.490,7.776,148.761
C00791=1152.416,250.945,-67.280,-177.488,7.779,148.760
C00792=1152.412,251.194,-67.307,-177.485,7.782,148.760
C00793=1152.408,251.443,-67.334,-177.482,7.784,148.760
C00794=1152.403,251.691,-67.362,-177.479,7.787,148.760
C00795=1152.399,251.939,-67.389,-177.477,7.790,148.760
C00796=1152.394,252.187,-67.417,-177.474,7.793,148.760
C00797=1152.390,252.436,-67.444,-177.472,7.795,148.760
C00798=1152.386,252.684,-67.472,-177.469,7.798,148.760
C00799=1152.381,252.933,-67.499,-177.466,7.801,148.760
C00800=1152.377,253.181,-67.527,-177.463,7.804,148.760
C00801=1152.372,253.430,-67.555,-177.460,7.807,148.760
C00802=1152.368,253.678,-67.583,-177.458,7.810,148.760
C00803=1152.364,253.927,-67.610,-177.455,7.813,148.760
C00804=1152.359,254.175,-67.638,-177.452,7.816,148.760
C00805=1152.355,254.424,-67.665,-177.449,7.819,148.759
C00806=1152.351,254.672,-67.693,-177.447,7.822,148.759
C00807=1152.346,254.921,-67.720,-177.444,7.825,148.759
C00808=1152.342,255.168,-67.748,-177.441,7.828,148.759
C00809=1152.338,255.418,-67.776,-177.439,7.830,148.759
C00810=1152.333,255.666,-67.804,-177.436,7.833,148.759
C00811=1152.328,255.914,-67.832,-177.433,7.836,148.759
C00812=1152.324,256.163,-67.859,-177.431,7.839,148.759
C00813=1152.320,256.411,-67.887,-177.428,7.842,148.759
C00814=1152.316,256.659,-67.915,-177.425,7.844,148.759
C00815=1152.311,256.908,-67.943,-177.422,7.847,148.759
C00816=1152.306,257.156,-67.971,-177.419,7.850,148.759
C00817=1152.303,257.405,-67.999,-177.417,7.853,148.759
C00818=1152.298,257.653,-68.026,-177.414,7.856,148.759
C00819=1152.294,257.902,-68.054,-177.411,7.859,148.759
C00820=1152.289,258.150,-68.082,-177.408,7.862,148.758
C00821=1152.285,258.398,-68.110,-177.406,7.865,148.758
C00822=1152.281,258.647,-68.137,-177.403,7.868,148.758
C00823=1152.276,258.895,-68.166,-177.400,7.871,148.758
C00824=1152.272,259.144,-68.194,-177.397,7.874,148.758
C00825=1152.268,259.392,-68.222,-177.395,7.877,148.758
C00826=1152.264,259.640,-68.250,-177.392,7.880,148.758
C00827=1152.259,259.888,-68.278,-177.390,7.882,148.758
C00828=1152.255,260.138,-68.306,-177.387,7.885,148.758
C00829=1152.250,260.385,-68.333,-177.384,7.888,148.758
C00830=1152.245,260.634,-68.362,-177.382,7.891,148.758
C00831=1152.242,260.882,-68.390,-177.379,7.894,148.758
C00832=1152.237,261.130,-68.418,-177.376,7.897,148.758
C00833=1152.232,261.404,-68.449,-177.373,7.901,148.758
C00834=1152.228,261.678,-68.480,-177.370,7.904,148.758
C00835=1152.223,261.951,-68.511,-177.367,7.907,148.758
C00836=1152.219,262.224,-68.542,-177.364,7.910,148.758
C00837=1152.214,262.472,-68.570,-177.361,7.913,148.758
C00838=1152.210,262.721,-68.599,-177.358,7.916,148.758
C00839=1152.205,262.969,-68.627,-177.355,7.919,148.758
C00840=1152.201,263.217,-68.655,-177.353,7.922,148.758
C00841=1152.197,263.465,-68.683,-177.350,7.925,148.758
C00842=1152.192,263.714,-68.712,-177.348,7.928,148.758
C00843=1152.188,263.962,-68.739,-177.345,7.931,148.758
C00844=1152.183,264.211,-68.768,-177.342,7.934,148.757
C00845=1152.179,264.459,-68.796,-177.339,7.937,148.757
C00846=1152.175,264.708,-68.825,-177.336,7.940,148.757
C00847=1152.171,264.956,-68.853,-177.334,7.943,148.757
C00848=1152.166,265.204,-68.881,-177.331,7.946,148.757
C00849=1152.162,265.453,-68.909,-177.329,7.949,148.757
C00850=1152.157,265.701,-68.938,-177.326,7.952,148.757
C00851=1152.153,265.949,-68.967,-177.323,7.955,148.757
C00852=1152.148,266.197,-68.995,-177.320,7.958,148.757
C00853=1152.145,266.446,-69.023,-177.318,7.961,148.757
C00854=1152.140,266.695,-69.052,-177.315,7.964,148.757
C00855=1152.135,266.942,-69.081,-177.312,7.967,148.757
C00856=1152.132,267.191,-69.109,-177.310,7.970,148.757
C00857=1152.126,267.439,-69.137,-177.307,7.973,148.757
C00858=1152.123,267.688,-69.166,-177.304,7.976,148.757
C00859=1152.119,267.936,-69.195,-177.301,7.979,148.757
C00860=1152.114,268.184,-69.223,-177.299,7.982,148.757
C00861=1152.110,268.433,-69.252,-177.296,7.985,148.757
C00862=1152.105,268.681,-69.281,-177.293,7.988,148.757
C00863=1152.101,268.929,-69.309,-177.291,7.991,148.757
C00864=1152.097,269.178,-69.338,-177.288,7.994,148.757
C00865=1152.092,269.426,-69.367,-177.285,7.997,148.757
C00866=1152.088,269.674,-69.395,-177.282,8.000,148.757
C00867=1152.084,269.923,-69.423,-177.280,8.003,148.757
C00868=1152.079,270.171,-69.453,-177.277,8.006,148.757
C00869=1152.075,270.419,-69.481,-177.275,8.009,148.757
C00870=1152.071,270.667,-69.510,-177.272,8.012,148.757
C00871=1152.066,270.916,-69.539,-177.269,8.015,148.757
C00872=1152.062,271.164,-69.567,-177.266,8.018,148.757
C00873=1152.058,271.412,-69.596,-177.264,8.021,148.757
C00874=1152.053,271.661,-69.625,-177.261,8.024,148.757
C00875=1152.049,271.909,-69.654,-177.258,8.027,148.757
C00876=1152.045,272.157,-69.682,-177.256,8.030,148.757
C00877=1152.041,272.405,-69.712,-177.253,8.033,148.757
C00878=1152.036,272.654,-69.740,-177.250,8.036,148.757
C00879=1152.031,272.902,-69.769,-177.248,8.039,148.757
C00880=1152.028,273.150,-69.798,-177.245,8.042,148.757
C00881=1152.024,273.399,-69.827,-177.242,8.045,148.757
C00882=1152.019,273.647,-69.856,-177.240,8.048,148.757
C00883=1152.014,273.895,-69.885,-177.237,8.051,148.757
C00884=1152.011,274.143,-69.914,-177.234,8.054,148.757
C00885=1152.007,274.391,-69.943,-177.232,8.057,148.757
C00886=1152.002,274.640,-69.972,-177.229,8.060,148.757
C00887=1151.998,274.889,-70.001,-177.226,8.063,148.757
C00888=1151.993,275.136,-70.030,-177.223,8.067,148.757
C00889=1151.989,275.385,-70.059,-177.220,8.070,148.757
C00890=1151.984,275.633,-70.089,-177.218,8.073,148.757
C00891=1151.981,275.881,-70.117,-177.215,8.076,148.757
C00892=1151.977,276.130,-70.146,-177.212,8.079,148.757
C00893=1151.972,276.378,-70.175,-177.210,8.082,148.757
C00894=1151.968,276.626,-70.205,-177.207,8.085,148.757
C00895=1151.963,276.874,-70.234,-177.205,8.088,148.757
C00896=1151.959,277.123,-70.264,-177.202,8.091,148.757
C00897=1151.955,277.371,-70.292,-177.199,8.094,148.757
C00898=1151.951,277.620,-70.322,-177.197,8.097,148.757
C00899=1151.946,277.867,-70.351,-177.194,8.100,148.757
C00900=1151.942,278.116,-70.380,-177.191,8.103,148.757
C00901=1151.938,278.363,-70.409,-177.188,8.106,148.757
C00902=1151.934,278.612,-70.439,-177.186,8.110,148.757
C00903=1151.929,278.861,-70.467,-177.183,8.113,148.757
C00904=1151.925,279.109,-70.497,-177.180,8.116,148.757
C00905=1151.921,279.357,-70.526,-177.178,8.119,148.757
C00906=1151.916,279.605,-70.555,-177.175,8.122,148.757
C00907=1151.912,279.853,-70.585,-177.172,8.125,148.757
C00908=1151.908,280.101,-70.614,-177.170,8.129,148.757
C00909=1151.904,280.350,-70.644,-177.167,8.132,148.757
C00910=1151.900,280.598,-70.673,-177.164,8.135,148.757
C00911=1151.895,280.846,-70.703,-177.162,8.138,148.757
C00912=1151.891,281.095,-70.733,-177.159,8.141,148.757
C00913=1151.886,281.343,-70.762,-177.156,8.144,148.757
C00914=1151.882,281.591,-70.792,-177.154,8.147,148.757
C00915=1151.878,281.839,-70.821,-177.151,8.151,148.757
C00916=1151.874,282.088,-70.851,-177.148,8.154,148.757
C00917=1151.870,282.336,-70.880,-177.146,8.157,148.757
C00918=1151.865,282.584,-70.909,-177.143,8.160,148.757
C00919=1151.861,282.832,-70.939,-177.140,8.163,148.757
C00920=1151.857,283.079,-70.969,-177.138,8.166,148.758
C00921=1151.852,283.328,-70.999,-177.135,8.169,148.757
C00922=1151.848,283.576,-71.028,-177.132,8.172,148.757
C00923=1151.843,283.825,-71.058,-177.130,8.175,148.758
C00924=1151.839,284.073,-71.087,-177.127,8.178,148.758
C00925=1151.835,284.321,-71.117,-177.124,8.182,148.758
C00926=1151.831,284.569,-71.146,-177.121,8.185,148.758
C00927=1151.826,284.817,-71.177,-177.119,8.188,148.758
C00928=1151.822,285.066,-71.206,-177.116,8.191,148.758
C00929=1151.818,285.314,-71.236,-177.114,8.194,148.758
C00930=1151.814,285.562,-71.265,-177.111,8.197,148.758
C00931=1151.810,285.810,-71.295,-177.109,8.201,148.758
C00932=1151.805,286.058,-71.325,-177.106,8.204,148.758
C00933=1151.801,286.307,-71.355,-177.103,8.207,148.758
C00934=1151.797,286.554,-71.385,-177.100,8.211,148.758
C00935=1151.793,286.803,-71.414,-177.097,8.214,148.758
C00936=1151.788,287.051,-71.444,-177.095,8.217,148.758
C00937=1151.784,287.327,-71.478,-177.092,8.220,148.758
C00938=1151.779,287.602,-71.511,-177.089,8.224,148.758
C00939=1151.774,287.877,-71.544,-177.086,8.228,148.758
C00940=1151.769,288.152,-71.577,-177.083,8.231,148.758
C00941=1151.765,288.401,-71.608,-177.080,8.234,148.758
C00942=1151.761,288.649,-71.637,-177.078,8.237,148.758
C00943=1151.757,288.897,-71.667,-177.075,8.241,148.758
C00944=1151.752,289.145,-71.697,-177.072,8.244,148.759
C00945=1151.748,289.393,-71.728,-177.070,8.247,148.759
C00946=1151.744,289.641,-71.757,-177.067,8.250,148.759
C00947=1151.740,289.889,-71.788,-177.065,8.253,148.759
C00948=1151.735,290.137,-71.817,-177.062,8.256,148.759
C00949=1151.732,290.385,-71.847,-177.060,8.259,148.759
C00950=1151.727,290.634,-71.878,-177.056,8.263,148.759
C00951=1151.723,290.882,-71.908,-177.054,8.266,148.759
C00952=1151.718,291.131,-71.938,-177.051,8.269,148.759
C00953=1151.715,291.378,-71.968,-177.049,8.272,148.759
C00954=1151.710,291.627,-71.998,-177.046,8.275,148.759
C00955=1151.706,291.874,-72.029,-177.043,8.278,148.759
C00956=1151.702,292.122,-72.059,-177.041,8.282,148.759
C00957=1151.697,292.371,-72.089,-177.038,8.285,148.759
C00958=1151.694,292.619,-72.119,-177.035,8.289,148.759
C00959=1151.689,292.867,-72.150,-177.032,8.292,148.759
C00960=1151.685,293.115,-72.179,-177.030,8.295,148.760
C00961=1151.680,293.363,-72.210,-177.027,8.298,148.760
C00962=1151.676,293.611,-72.240,-177.025,8.301,148.760
C00963=1151.672,293.860,-72.271,-177.022,8.305,148.760
C00964=1151.668,294.108,-72.301,-177.019,8.308,148.760
C00965=1151.664,294.356,-72.332,-177.017,8.311,148.760
C00966=1151.660,294.603,-72.362,-177.014,8.314,148.760
C00967=1151.655,294.852,-72.392,-177.012,8.317,148.760
C00968=1151.652,295.100,-72.423,-177.009,8.321,148.760
C00969=1151.647,295.348,-72.453,-177.006,8.324,148.760
C00970=1151.643,295.596,-72.483,-177.004,8.328,148.760
C00971=1151.638,295.844,-72.514,-177.001,8.331,148.760
C00972=1151.634,296.093,-72.545,-176.998,8.334,148.760
C00973=1151.630,296.341,-72.575,-176.996,8.337,148.760
C00974=1151.626,296.589,-72.606,-176.993,8.341,148.761
C00975=1151.622,296.836,-72.636,-176.990,8.344,148.761
C00976=1151.618,297.085,-72.667,-176.988,8.347,148.761
C00977=1151.613,297.333,-72.698,-176.985,8.350,148.761
C00978=1151.609,297.581,-72.728,-176.983,8.353,148.761
C00979=1151.605,297.829,-72.759,-176.980,8.357,148.761
C00980=1151.601,298.077,-72.790,-176.977,8.360,148.761
C00981=1151.597,298.325,-72.820,-176.975,8.364,148.761
C00982=1151.592,298.573,-72.851,-176.972,8.367,148.761
C00983=1151.588,298.822,-72.882,-176.970,8.370,148.761
C00984=1151.584,299.069,-72.912,-176.967,8.373,148.761
C00985=1151.580,299.317,-72.943,-176.964,8.377,148.762
C00986=1151.576,299.566,-72.974,-176.961,8.380,148.762
C00987=1151.572,299.813,-73.004,-176.959,8.383,148.762
C00988=1151.567,300.061,-73.035,-176.957,8.386,148.762
C00989=1151.563,300.310,-73.066,-176.954,8.389,148.762
C00990=1151.559,300.558,-73.097,-176.951,8.393,148.762
C00991=1151.555,300.806,-73.127,-176.948,8.396,148.762
C00992=1151.551,301.054,-73.158,-176.946,8.400,148.762
C00993=1151.546,301.302,-73.189,-176.943,8.403,148.762
C00994=1151.542,301.550,-73.220,-176.940,8.407,148.762
C00995=1151.538,301.798,-73.251,-176.938,8.410,148.763
C00996=1151.534,302.046,-73.281,-176.935,8.413,148.763
C00997=1151.529,302.294,-73.312,-176.933,8.416,148.763
C00998=1151.525,302.543,-73.343,-176.930,8.419,148.763
C00999=1151.521,302.791,-73.374,-176.927,8.423,148.763
C01000=1151.517,303.039,-73.406,-176.925,8.427,148.763
C01001=1151.512,303.287,-73.437,-176.922,8.429,148.763
C01002=1151.508,303.534,-73.467,-176.920,8.433,148.763
C01003=1151.504,303.783,-73.498,-176.917,8.437,148.764
C01004=1151.500,304.030,-73.530,-176.914,8.440,148.763
C01005=1151.496,304.279,-73.561,-176.912,8.443,148.764
C01006=1151.491,304.527,-73.591,-176.909,8.446,148.764
C01007=1151.487,304.774,-73.623,-176.907,8.449,148.764
C01008=1151.483,305.023,-73.654,-176.904,8.453,148.764
C01009=1151.478,305.271,-73.685,-176.901,8.456,148.764
C01010=1151.475,305.519,-73.717,-176.899,8.460,148.764
C01011=1151.470,305.767,-73.747,-176.896,8.463,148.764
C01012=1151.466,306.015,-73.779,-176.893,8.467,148.764
C01013=1151.462,306.263,-73.810,-176.891,8.470,148.765
C01014=1151.457,306.511,-73.841,-176.888,8.473,148.765
C01015=1151.454,306.759,-73.873,-176.886,8.476,148.765
C01016=1151.449,307.007,-73.903,-176.883,8.480,148.765
C01017=1151.445,307.255,-73.935,-176.880,8.483,148.765
C01018=1151.441,307.503,-73.966,-176.878,8.486,148.765
C01019=1151.437,307.751,-73.998,-176.875,8.490,148.765
C01020=1151.432,307.999,-74.029,-176.872,8.494,148.766
C01021=1151.429,308.247,-74.060,-176.870,8.497,148.765
C01022=1151.424,308.495,-74.091,-176.867,8.500,148.766
C01023=1151.420,308.743,-74.123,-176.865,8.503,148.766
C01024=1151.416,308.991,-74.154,-176.862,8.507,148.766
C01025=1151.412,309.239,-74.186,-176.859,8.510,148.766
C01026=1151.408,309.486,-74.217,-176.857,8.514,148.766
C01027=1151.404,309.735,-74.248,-176.855,8.517,148.766
C01028=1151.400,309.983,-74.280,-176.851,8.521,148.766
C01029=1151.395,310.231,-74.311,-176.849,8.524,148.767
C01030=1151.392,310.479,-74.343,-176.847,8.527,148.767
C01031=1151.387,310.726,-74.374,-176.843,8.531,148.767
C01032=1151.383,310.975,-74.406,-176.841,8.534,148.767
C01033=1151.378,311.222,-74.437,-176.839,8.538,148.767
C01034=1151.375,311.470,-74.469,-176.836,8.541,148.767
C01035=1151.370,311.718,-74.501,-176.833,8.545,148.767
C01036=1151.366,311.966,-74.532,-176.831,8.548,148.768
C01037=1151.362,312.214,-74.564,-176.828,8.551,148.768
C01038=1151.358,312.462,-74.595,-176.826,8.554,148.768
C01039=1151.354,312.710,-74.628,-176.823,8.558,148.768
C01040=1151.349,312.958,-74.658,-176.820,8.561,148.768
C01041=1151.345,313.236,-74.694,-176.817,8.566,148.768
C01042=1151.340,313.513,-74.730,-176.815,8.570,148.769
C01043=1151.336,313.791,-74.765,-176.812,8.573,148.769
C01044=1151.331,314.069,-74.801,-176.809,8.577,148.769
C01045=1151.327,314.316,-74.833,-176.806,8.581,148.769
C01046=1151.323,314.565,-74.864,-176.804,8.584,148.769
C01047=1151.318,314.812,-74.895,-176.801,8.587,148.769
C01048=1151.314,315.060,-74.928,-176.799,8.590,148.769
C01049=1151.310,315.308,-74.960,-176.796,8.594,148.770
C01050=1151.306,315.556,-74.991,-176.793,8.598,148.770
C01051=1151.302,315.804,-75.023,-176.791,8.601,148.770
C01052=1151.298,316.052,-75.056,-176.788,8.605,148.770
C01053=1151.294,316.300,-75.087,-176.785,8.608,148.770
C01054=1151.290,316.547,-75.119,-176.783,8.611,148.770
C01055=1151.285,316.796,-75.151,-176.780,8.615,148.771
C01056=1151.282,317.044,-75.183,-176.778,8.619,148.771
C01057=1151.277,317.291,-75.215,-176.775,8.622,148.771
C01058=1151.273,317.539,-75.247,-176.773,8.625,148.771
C01059=1151.269,317.788,-75.279,-176.770,8.629,148.771
C01060=1151.265,318.035,-75.310,-176.768,8.632,148.771
C01061=1151.261,318.283,-75.343,-176.765,8.635,148.772
C01062=1151.257,318.531,-75.375,-176.762,8.639,148.772
C01063=1151.253,318.779,-75.408,-176.760,8.642,148.772
C01064=1151.248,319.026,-75.439,-176.757,8.646,148.772
C01065=1151.245,319.274,-75.471,-176.754,8.650,148.772
C01066=1151.240,319.523,-75.504,-176.752,8.653,148.772
C01067=1151.237,319.771,-75.535,-176.750,8.656,148.773
C01068=1151.232,320.018,-75.568,-176.747,8.660,148.773
C01069=1151.228,320.266,-75.600,-176.744,8.663,148.773
C01070=1151.224,320.514,-75.633,-176.742,8.667,148.773
C01071=1151.220,320.762,-75.664,-176.739,8.671,148.773
C01072=1151.216,321.010,-75.696,-176.737,8.674,148.773
C01073=1151.211,321.257,-75.729,-176.734,8.677,148.774
C01074=1151.208,321.505,-75.761,-176.731,8.681,148.774
C01075=1151.203,321.754,-75.793,-176.729,8.685,148.774
C01076=1151.200,322.001,-75.826,-176.727,8.688,148.774
C01077=1151.195,322.249,-75.858,-176.723,8.692,148.774
C01078=1151.191,322.498,-75.891,-176.721,8.695,148.774
C01079=1151.187,322.744,-75.923,-176.719,8.698,148.775
C01080=1151.183,322.993,-75.955,-176.716,8.702,148.775
C01081=1151.179,323.241,-75.987,-176.713,8.706,148.775
C01082=1151.175,323.489,-76.020,-176.711,8.710,148.775
C01083=1151.171,323.737,-76.052,-176.708,8.713,148.775
C01084=1151.167,323.984,-76.085,-176.706,8.716,148.776
C01085=1151.163,324.232,-76.117,-176.703,8.720,148.776
C01086=1151.158,324.479,-76.150,-176.701,8.724,148.776
C01087=1151.154,324.728,-76.182,-176.698,8.727,148.776
C01088=1151.151,324.975,-76.215,-176.695,8.731,148.776
C01089=1151.146,325.224,-76.247,-176.693,8.734,148.777
C01090=1151.142,325.471,-76.281,-176.690,8.737,148.777
C01091=1151.138,325.719,-76.312,-176.687,8.741,148.777
C01092=1151.134,325.967,-76.346,-176.685,8.745,148.777
C01093=1151.130,326.215,-76.377,-176.682,8.749,148.777
C01094=1151.126,326.462,-76.410,-176.680,8.752,148.778
C01095=1151.121,326.710,-76.443,-176.678,8.755,148.778
C01096=1151.117,326.958,-76.476,-176.675,8.759,148.778
C01097=1151.114,327.206,-76.508,-176.672,8.763,148.778
C01098=1151.109,327.454,-76.541,-176.670,8.766,148.778
C01099=1151.105,327.702,-76.574,-176.667,8.770,148.779
C01100=1151.101,327.950,-76.606,-176.665,8.773,148.779
C01101=1151.097,328.197,-76.639,-176.662,8.777,148.779
C01102=1151.093,328.445,-76.672,-176.660,8.781,148.779
C01103=1151.089,328.694,-76.705,-176.657,8.784,148.779
C01104=1151.085,328.941,-76.737,-176.654,8.788,148.780
C01105=1151.081,329.189,-76.770,-176.652,8.791,148.780
C01106=1151.077,329.436,-76.803,-176.650,8.795,148.780
C01107=1151.073,329.685,-76.836,-176.647,8.799,148.780
C01108=1151.068,329.932,-76.869,-176.645,8.802,148.781
C01109=1151.065,330.180,-76.902,-176.642,8.806,148.781
C01110=1151.061,330.428,-76.935,-176.639,8.809,148.781
C01111=1151.057,330.675,-76.968,-176.637,8.813,148.781
C01112=1151.052,330.924,-77.000,-176.634,8.817,148.781
C01113=1151.048,331.171,-77.034,-176.632,8.820,148.782
C01114=1151.044,331.419,-77.067,-176.629,8.824,148.782
C01115=1151.040,331.667,-77.100,-176.627,8.827,148.782
C01116=1151.037,331.914,-77.132,-176.624,8.831,148.782
C01117=1151.032,332.162,-77.166,-176.621,8.835,148.782
C01118=1151.028,332.410,-77.199,-176.619,8.838,148.783
C01119=1151.024,332.658,-77.232,-176.616,8.842,148.783
C01120=1151.020,332.905,-77.265,-176.614,8.845,148.783
C01121=1151.016,333.154,-77.297,-176.611,8.849,148.783
C01122=1151.011,333.401,-77.331,-176.609,8.853,148.784
C01123=1151.007,333.649,-77.364,-176.606,8.856,148.784
C01124=1151.003,333.897,-77.397,-176.603,8.860,148.784
C01125=1150.999,334.145,-77.430,-176.601,8.863,148.784
C01126=1150.995,334.392,-77.463,-176.598,8.867,148.784
C01127=1150.991,334.639,-77.497,-176.596,8.871,148.785
C01128=1150.987,334.887,-77.530,-176.593,8.875,148.785
C01129=1150.983,335.136,-77.564,-176.591,8.878,148.785
C01130=1150.979,335.383,-77.597,-176.589,8.882,148.785
C01131=1150.975,335.631,-77.630,-176.586,8.886,148.786
C01132=1150.971,335.879,-77.663,-176.583,8.889,148.786
C01133=1150.967,336.126,-77.696,-176.581,8.893,148.786
C01134=1150.963,336.374,-77.730,-176.578,8.896,148.786
C01135=1150.959,336.622,-77.763,-176.575,8.900,148.787
C01136=1150.955,336.869,-77.797,-176.573,8.904,148.787
C01137=1150.951,337.117,-77.830,-176.571,8.907,148.787
C01138=1150.947,337.365,-77.863,-176.568,8.911,148.787
C01139=1150.943,337.613,-77.896,-176.565,8.914,148.787
C01140=1150.939,337.861,-77.930,-176.563,8.919,148.788
C01141=1150.935,338.108,-77.963,-176.561,8.922,148.788
C01142=1150.931,338.355,-77.997,-176.558,8.926,148.788
C01143=1150.927,338.603,-78.030,-176.555,8.929,148.789
C01144=1150.922,338.852,-78.064,-176.553,8.933,148.789
C01145=1150.918,339.131,-78.101,-176.550,8.938,148.789
C01146=1150.914,339.412,-78.139,-176.547,8.942,148.789
C01147=1150.908,339.692,-78.177,-176.544,8.946,148.790
C01148=1150.904,339.972,-78.215,-176.541,8.950,148.790
C01149=1150.901,340.219,-78.249,-176.539,8.953,148.790
C01150=1150.896,340.467,-78.283,-176.536,8.957,148.790
C01151=1150.892,340.716,-78.316,-176.534,8.961,148.791
C01152=1150.888,340.963,-78.350,-176.531,8.965,148.791
C01153=1150.884,341.210,-78.384,-176.529,8.968,148.791
C01154=1150.880,341.458,-78.418,-176.526,8.973,148.792
C01155=1150.876,341.706,-78.451,-176.524,8.976,148.792
C01156=1150.872,341.953,-78.485,-176.521,8.980,148.792
C01157=1150.868,342.201,-78.519,-176.519,8.983,148.792
C01158=1150.864,342.449,-78.553,-176.516,8.987,148.792
C01159=1150.859,342.696,-78.586,-176.514,8.991,148.793
C01160=1150.856,342.944,-78.620,-176.511,8.995,148.793
C01161=1150.852,343.192,-78.654,-176.509,8.998,148.793
C01162=1150.847,343.439,-78.688,-176.506,9.001,148.794
C01163=1150.843,343.687,-78.721,-176.503,9.006,148.794
C01164=1150.840,343.935,-78.755,-176.501,9.009,148.794
C01165=1150.835,344.183,-78.789,-176.499,9.013,148.794
C01166=1150.831,344.430,-78.823,-176.496,9.017,148.795
C01167=1150.828,344.678,-78.857,-176.493,9.021,148.795
C01168=1150.823,344.926,-78.891,-176.491,9.024,148.795
C01169=1150.819,345.173,-78.925,-176.489,9.028,148.796
C01170=1150.816,345.421,-78.959,-176.486,9.032,148.796
C01171=1150.811,345.669,-78.993,-176.483,9.036,148.796
C01172=1150.808,345.916,-79.027,-176.481,9.039,148.796
C01173=1150.803,346.163,-79.061,-176.478,9.043,148.796
C01174=1150.799,346.412,-79.095,-176.476,9.047,148.797
C01175=1150.795,346.659,-79.129,-176.473,9.051,148.797
C01176=1150.792,346.907,-79.163,-176.470,9.055,148.797
C01177=1150.788,347.154,-79.197,-176.468,9.058,148.798
C01178=1150.783,347.402,-79.231,-176.466,9.062,148.798
C01179=1150.780,347.650,-79.265,-176.463,9.066,148.798
C01180=1150.775,347.897,-79.300,-176.460,9.070,148.799
C01181=1150.771,348.144,-79.334,-176.458,9.073,148.799
C01182=1150.767,348.392,-79.368,-176.456,9.077,148.799
C01183=1150.763,348.640,-79.402,-176.453,9.081,148.799
C01184=1150.760,348.888,-79.437,-176.450,9.085,148.800
C01185=1150.755,349.135,-79.470,-176.448,9.088,148.800
C01186=1150.751,349.383,-79.505,-176.446,9.093,148.800
C01187=1150.748,349.631,-79.539,-176.443,9.096,148.801
C01188=1150.743,349.878,-79.573,-176.440,9.100,148.801
C01189=1150.740,350.126,-79.608,-176.438,9.103,148.801
C01190=1150.735,350.373,-79.642,-176.435,9.108,148.801
C01191=1150.731,350.620,-79.676,-176.433,9.111,148.802
C01192=1150.727,350.869,-79.711,-176.431,9.115,148.802
C01193=1150.723,351.116,-79.745,-176.428,9.119,148.802
C01194=1150.720,351.364,-79.780,-176.425,9.123,148.803
C01195=1150.715,351.611,-79.814,-176.423,9.127,148.803
C01196=1150.712,351.859,-79.848,-176.421,9.130,148.803
C01197=1150.707,352.106,-79.883,-176.418,9.134,148.803
C01198=1150.703,352.355,-79.918,-176.415,9.138,148.804
C01199=1150.699,352.602,-79.951,-176.413,9.142,148.804
C01200=1150.696,352.849,-79.987,-176.411,9.145,148.804
C01201=1150.692,353.096,-80.021,-176.408,9.149,148.805
C01202=1150.688,353.344,-80.056,-176.405,9.154,148.805
C01203=1150.683,353.592,-80.090,-176.403,9.157,148.805
C01204=1150.680,353.840,-80.124,-176.400,9.161,148.806
C01205=1150.676,354.087,-80.159,-176.398,9.165,148.806
C01206=1150.672,354.335,-80.194,-176.395,9.169,148.806
C01207=1150.667,354.582,-80.229,-176.393,9.172,148.806
C01208=1150.664,354.830,-80.263,-176.390,9.177,148.807
C01209=1150.660,355.077,-80.298,-176.388,9.180,148.807
C01210=1150.656,355.325,-80.332,-176.386,9.184,148.808
C01211=1150.652,355.572,-80.367,-176.383,9.188,148.808
C01212=1150.648,355.820,-80.402,-176.380,9.192,148.808
C01213=1150.644,356.067,-80.436,-176.378,9.196,148.809
C01214=1150.640,356.315,-80.472,-176.376,9.199,148.809
C01215=1150.637,356.563,-80.506,-176.373,9.203,148.809
C01216=1150.632,356.810,-80.541,-176.370,9.208,148.809
C01217=1150.628,357.058,-80.576,-176.368,9.211,148.810
C01218=1150.624,357.305,-80.611,-176.365,9.215,148.810
C01219=1150.620,357.552,-80.646,-176.363,9.219,148.810
C01220=1150.617,357.800,-80.680,-176.360,9.223,148.811
C01221=1150.612,358.048,-80.715,-176.358,9.227,148.811
C01222=1150.609,358.295,-80.750,-176.355,9.230,148.811
C01223=1150.604,358.543,-80.785,-176.352,9.235,148.812
C01224=1150.600,358.790,-80.820,-176.351,9.238,148.812
C01225=1150.597,359.038,-80.855,-176.348,9.242,148.812
C01226=1150.593,359.285,-80.890,-176.345,9.247,148.813
C01227=1150.589,359.533,-80.925,-176.343,9.250,148.813
C01228=1150.585,359.780,-80.960,-176.340,9.254,148.813
C01229=1150.581,360.028,-80.995,-176.337,9.258,148.814
C01230=1150.577,360.275,-81.030,-176.335,9.262,148.814
C01231=1150.573,360.523,-81.065,-176.332,9.266,148.814
C01232=1150.569,360.770,-81.100,-176.330,9.270,148.815
C01233=1150.565,361.018,-81.136,-176.327,9.273,148.815
C01234=1150.561,361.266,-81.171,-176.325,9.278,148.815
C01235=1150.557,361.513,-81.206,-176.322,9.282,148.816
C01236=1150.554,361.760,-81.241,-176.320,9.285,148.816
C01237=1150.550,362.008,-81.276,-176.317,9.290,148.816
C01238=1150.546,362.255,-81.311,-176.314,9.294,148.816
C01239=1150.542,362.502,-81.346,-176.312,9.298,148.817
C01240=1150.538,362.750,-81.381,-176.310,9.301,148.817
C01241=1150.535,362.998,-81.417,-176.307,9.305,148.817
C01242=1150.530,363.245,-81.452,-176.304,9.310,148.818
C01243=1150.527,363.492,-81.487,-176.302,9.313,148.818
C01244=1150.523,363.740,-81.522,-176.299,9.317,148.819
C01245=1150.518,363.987,-81.557,-176.296,9.322,148.819
C01246=1150.515,364.235,-81.593,-176.294,9.326,148.819
C01247=1150.510,364.482,-81.629,-176.292,9.329,148.819
C01248=1150.507,364.730,-81.665,-176.289,9.333,148.820
C01249=1150.503,365.014,-81.704,-176.286,9.339,148.820
C01250=1150.498,365.296,-81.745,-176.283,9.343,148.821
C01251=1150.493,365.580,-81.785,-176.280,9.347,148.821
C01252=1150.489,365.863,-81.826,-176.277,9.352,148.822
C01253=1150.485,366.111,-81.862,-176.274,9.356,148.822
C01254=1150.481,366.357,-81.897,-176.272,9.360,148.822
C01255=1150.477,366.605,-81.932,-176.269,9.364,148.823
C01256=1150.474,366.852,-81.968,-176.267,9.368,148.823
C01257=1150.469,367.100,-82.004,-176.264,9.372,148.823
C01258=1150.465,367.348,-82.040,-176.262,9.376,148.824
C01259=1150.461,367.594,-82.075,-176.259,9.380,148.824
C01260=1150.458,367.842,-82.110,-176.257,9.385,148.824
C01261=1150.454,368.089,-82.146,-176.254,9.389,148.825
C01262=1150.450,368.337,-82.182,-176.252,9.392,148.825
C01263=1150.446,368.585,-82.218,-176.250,9.397,148.826
C01264=1150.442,368.832,-82.253,-176.247,9.401,148.826
C01265=1150.438,369.079,-82.288,-176.244,9.405,148.826
C01266=1150.434,369.326,-82.325,-176.242,9.409,148.827
C01267=1150.430,369.574,-82.361,-176.239,9.413,148.827
C01268=1150.426,369.821,-82.396,-176.237,9.417,148.827
C01269=1150.423,370.069,-82.432,-176.234,9.422,148.828
C01270=1150.418,370.317,-82.468,-176.232,9.425,148.828
C01271=1150.415,370.564,-82.504,-176.230,9.429,148.829
C01272=1150.411,370.811,-82.540,-176.227,9.434,148.829
C01273=1150.407,371.058,-82.575,-176.225,9.438,148.830
C01274=1150.403,371.306,-82.611,-176.223,9.442,148.830
C01275=1150.399,371.553,-82.647,-176.220,9.446,148.830
C01276=1150.396,371.800,-82.683,-176.218,9.450,148.831
C01277=1150.391,372.048,-82.719,-176.216,9.454,148.831
C01278=1150.388,372.295,-82.755,-176.213,9.458,148.832
C01279=1150.384,372.543,-82.790,-176.211,9.463,148.832
C01280=1150.380,372.790,-82.827,-176.209,9.466,148.833
C01281=1150.376,373.037,-82.863,-176.206,9.471,148.833
C01282=1150.372,373.285,-82.899,-176.204,9.475,148.834
C01283=1150.368,373.532,-82.935,-176.202,9.479,148.834
C01284=1150.365,373.780,-82.971,-176.200,9.483,148.835
C01285=1150.361,374.027,-83.007,-176.198,9.487,148.835
C01286=1150.357,374.274,-83.043,-176.195,9.491,148.835
C01287=1150.353,374.522,-83.079,-176.193,9.496,148.836
C01288=1150.349,374.769,-83.115,-176.191,9.499,148.837
C01289=1150.345,375.017,-83.151,-176.189,9.504,148.837
C01290=1150.342,375.264,-83.188,-176.187,9.508,148.838
C01291=1150.338,375.511,-83.223,-176.185,9.512,148.838
C01292=1150.334,375.758,-83.260,-176.183,9.516,148.839
C01293=1150.330,376.006,-83.296,-176.181,9.520,148.839
C01294=1150.326,376.253,-83.333,-176.179,9.524,148.840
C01295=1150.322,376.501,-83.368,-176.177,9.528,148.840
C01296=1150.318,376.748,-83.405,-176.175,9.532,148.841
C01297=1150.315,376.995,-83.441,-176.173,9.536,148.841
C01298=1150.311,377.242,-83.477,-176.172,9.540,148.842
C01299=1150.307,377.489,-83.514,-176.170,9.544,148.842
C01300=1150.303,377.737,-83.550,-176.168,9.548,148.843
C01301=1150.299,377.984,-83.587,-176.167,9.552,148.844
C01302=1150.295,378.232,-83.622,-176.165,9.557,148.844
C01303=1150.291,378.479,-83.659,-176.163,9.561,148.845
C01304=1150.288,378.726,-83.695,-176.161,9.564,148.845
C01305=1150.283,378.974,-83.731,-176.160,9.568,148.846
C01306=1150.280,379.221,-83.768,-176.158,9.572,148.847
C01307=1150.276,379.468,-83.805,-176.157,9.576,148.847
C01308=1150.271,379.716,-83.841,-176.155,9.580,148.848
C01309=1150.268,379.962,-83.877,-176.154,9.584,148.849
C01310=1150.264,380.210,-83.914,-176.153,9.588,148.849
C01311=1150.261,380.457,-83.950,-176.151,9.592,148.850
C01312=1150.257,380.705,-83.987,-176.150,9.596,148.850
C01313=1150.253,380.952,-84.023,-176.149,9.600,148.851
C01314=1150.249,381.199,-84.060,-176.147,9.604,148.852
C01315=1150.245,381.446,-84.097,-176.146,9.607,148.852
C01316=1150.241,381.694,-84.133,-176.145,9.611,148.853
C01317=1150.237,381.941,-84.169,-176.144,9.615,148.854
C01318=1150.233,382.188,-84.206,-176.143,9.618,148.855
C01319=1150.229,382.435,-84.243,-176.142,9.622,148.855
C01320=1150.226,382.682,-84.279,-176.141,9.627,148.856
C01321=1150.221,382.930,-84.315,-176.140,9.630,148.857
C01322=1150.218,383.178,-84.352,-176.139,9.633,148.857
C01323=1150.215,383.425,-84.389,-176.138,9.637,148.858
C01324=1150.211,383.672,-84.425,-176.138,9.641,148.859
C01325=1150.206,383.919,-84.462,-176.137,9.644,148.860
C01326=1150.202,384.166,-84.499,-176.136,9.648,148.861
C01327=1150.199,384.413,-84.535,-176.136,9.652,148.861
C01328=1150.195,384.660,-84.572,-176.135,9.655,148.862
C01329=1150.191,384.908,-84.610,-176.135,9.658,148.863
C01330=1150.188,385.156,-84.645,-176.134,9.662,148.864
C01331=1150.184,385.403,-84.682,-176.134,9.665,148.864
C01332=1150.180,385.650,-84.719,-176.134,9.668,148.865
C01333=1150.175,385.897,-84.756,-176.134,9.671,148.866
C01334=1150.172,386.144,-84.792,-176.134,9.675,148.867
C01335=1150.169,386.392,-84.829,-176.133,9.678,148.868
C01336=1150.164,386.639,-84.866,-176.134,9.681,148.868
C01337=1150.160,386.887,-84.903,-176.133,9.684,148.869
C01338=1150.157,387.133,-84.939,-176.133,9.687,148.870
C01339=1150.153,387.381,-84.976,-176.133,9.691,148.871
C01340=1150.149,387.628,-85.013,-176.133,9.693,148.872
C01341=1150.145,387.876,-85.050,-176.134,9.696,148.872
C01342=1150.142,388.123,-85.086,-176.133,9.699,148.873
C01343=1150.138,388.370,-85.123,-176.134,9.702,148.874
C01344=1150.134,388.617,-85.160,-176.134,9.705,148.875
C01345=1150.130,388.864,-85.197,-176.135,9.708,148.876
C01346=1150.127,389.112,-85.234,-176.135,9.711,148.877
C01347=1150.123,389.359,-85.270,-176.135,9.714,148.878
C01348=1150.119,389.606,-85.307,-176.135,9.717,148.878
C01349=1150.115,389.853,-85.344,-176.136,9.720,148.879
C01350=1150.111,390.101,-85.381,-176.136,9.723,148.880
C01351=1150.108,390.348,-85.418,-176.137,9.724,148.881
C01352=1150.104,390.595,-85.454,-176.137,9.727,148.882
C01353=1150.099,390.882,-85.497,-176.138,9.730,148.883
C01354=1150.095,391.168,-85.540,-176.139,9.733,148.884
C01355=1150.090,391.454,-85.582,-176.139,9.736,148.884
C01356=1150.085,391.741,-85.626,-176.140,9.739,148.886
C01357=1150.083,391.988,-85.662,-176.141,9.742,148.886
C01358=1150.079,392.236,-85.699,-176.141,9.745,148.887
C01359=1150.074,392.483,-85.736,-176.142,9.747,148.888
C01360=1150.070,392.730,-85.773,-176.143,9.750,148.889
C01361=1150.066,392.977,-85.810,-176.144,9.752,148.890
C01362=1150.063,393.225,-85.846,-176.144,9.755,148.891
C01363=1150.059,393.472,-85.883,-176.145,9.757,148.891
C01364=1150.055,393.719,-85.920,-176.146,9.760,148.892
C01365=1150.051,393.966,-85.957,-176.147,9.762,148.893
C01366=1150.047,394.213,-85.994,-176.147,9.764,148.894
C01367=1150.044,394.461,-86.031,-176.148,9.766,148.895
C01368=1150.040,394.708,-86.067,-176.149,9.768,148.896
C01369=1150.036,394.955,-86.104,-176.150,9.771,148.896
C01370=1150.032,395.202,-86.142,-176.151,9.773,148.897
C01371=1150.028,395.449,-86.178,-176.152,9.775,148.898
C01372=1150.025,395.697,-86.216,-176.153,9.778,148.899
C01373=1150.021,395.944,-86.252,-176.154,9.780,148.900
C01374=1150.017,396.191,-86.289,-176.155,9.782,148.901
C01375=1150.013,396.438,-86.326,-176.156,9.784,148.902
C01376=1150.009,396.685,-86.362,-176.157,9.786,148.902
C01377=1150.006,396.933,-86.400,-176.157,9.789,148.903
C01378=1150.002,397.181,-86.437,-176.158,9.791,148.904
C01379=1149.998,397.427,-86.473,-176.159,9.793,148.905
C01380=1149.994,397.675,-86.510,-176.160,9.795,148.906
C01381=1149.991,397.923,-86.547,-176.162,9.797,148.906
C01382=1149.987,398.170,-86.584,-176.163,9.799,148.907
C01383=1149.983,398.416,-86.621,-176.164,9.801,148.908
C01384=1149.979,398.663,-86.658,-176.164,9.803,148.909
C01385=1149.975,398.910,-86.694,-176.166,9.805,148.910
C01386=1149.972,399.158,-86.732,-176.167,9.807,148.910
C01387=1149.968,399.405,-86.769,-176.168,9.809,148.911
C01388=1149.964,399.653,-86.805,-176.169,9.811,148.912
C01389=1149.960,399.900,-86.842,-176.170,9.813,148.913
C01390=1149.955,400.147,-86.879,-176.171,9.815,148.914
C01391=1149.952,400.395,-86.916,-176.172,9.817,148.914
C01392=1149.949,400.642,-86.953,-176.173,9.819,148.915
C01393=1149.944,400.889,-86.989,-176.174,9.821,148.916
C01394=1149.940,401.136,-87.026,-176.175,9.823,148.917
C01395=1149.937,401.383,-87.064,-176.176,9.825,148.918
C01396=1149.933,401.631,-87.101,-176.177,9.827,148.918
C01397=1149.929,401.878,-87.138,-176.178,9.829,148.919
C01398=1149.926,402.125,-87.174,-176.179,9.831,148.920
C01399=1149.922,402.372,-87.211,-176.180,9.833,148.921
C01400=1149.917,402.619,-87.248,-176.181,9.835,148.922
C01401=1149.914,402.867,-87.285,-176.182,9.837,148.922
C01402=1149.910,403.114,-87.322,-176.183,9.839,148.923
C01403=1149.906,403.361,-87.359,-176.184,9.841,148.924
C01404=1149.902,403.608,-87.395,-176.185,9.843,148.925
C01405=1149.899,403.856,-87.432,-176.186,9.845,148.925
C01406=1149.895,404.103,-87.470,-176.187,9.846,148.926
C01407=1149.891,404.350,-87.507,-176.188,9.848,148.927
C01408=1149.887,404.597,-87.544,-176.189,9.850,148.928
C01409=1149.883,404.844,-87.581,-176.190,9.852,148.928
C01410=1149.880,405.092,-87.617,-176.191,9.854,148.929
C01411=1149.876,405.339,-87.654,-176.192,9.856,148.930
C01412=1149.872,405.586,-87.691,-176.193,9.857,148.931
C01413=1149.868,405.833,-87.728,-176.194,9.860,148.931
C01414=1149.864,406.081,-87.765,-176.194,9.861,148.932
C01415=1149.860,406.329,-87.802,-176.195,9.863,148.933
C01416=1149.856,406.576,-87.839,-176.196,9.865,148.934
C01417=1149.853,406.822,-87.876,-176.197,9.867,148.934
C01418=1149.849,407.069,-87.913,-176.198,9.869,148.935
C01419=1149.845,407.317,-87.950,-176.200,9.870,148.936
C01420=1149.841,407.564,-87.987,-176.200,9.872,148.936
C01421=1149.837,407.811,-88.023,-176.201,9.874,148.937
C01422=1149.833,408.059,-88.060,-176.202,9.876,148.938
C01423=1149.830,408.305,-88.097,-176.203,9.878,148.939
C01424=1149.826,408.553,-88.134,-176.204,9.880,148.939
C01425=1149.822,408.801,-88.171,-176.205,9.882,148.940
C01426=1149.818,409.048,-88.208,-176.206,9.883,148.941
C01427=1149.814,409.294,-88.245,-176.206,9.885,148.942
C01428=1149.810,409.542,-88.282,-176.207,9.887,148.942
C01429=1149.808,409.789,-88.319,-176.208,9.889,148.943
C01430=1149.803,410.036,-88.355,-176.209,9.891,148.944
C01431=1149.799,410.283,-88.392,-176.210,9.893,148.944
C01432=1149.795,410.531,-88.429,-176.211,9.894,148.945
C01433=1149.792,410.779,-88.466,-176.211,9.896,148.946
C01434=1149.788,411.026,-88.503,-176.212,9.898,148.947
C01435=1149.784,411.273,-88.540,-176.213,9.900,148.947
C01436=1149.781,411.519,-88.577,-176.214,9.902,148.948
C01437=1149.776,411.766,-88.614,-176.214,9.904,148.949
C01438=1149.773,412.014,-88.651,-176.215,9.906,148.949
C01439=1149.769,412.261,-88.688,-176.216,9.908,148.950
C01440=1149.765,412.509,-88.725,-176.216,9.910,148.951
C01441=1149.761,412.756,-88.762,-176.217,9.912,148.951
C01442=1149.757,413.003,-88.799,-176.218,9.914,148.952
C01443=1149.754,413.251,-88.835,-176.219,9.915,148.953
C01444=1149.750,413.498,-88.872,-176.219,9.917,148.953
C01445=1149.746,413.744,-88.910,-176.220,9.919,148.954
C01446=1149.742,413.992,-88.947,-176.221,9.921,148.955
C01447=1149.738,414.239,-88.984,-176.222,9.923,148.956
C01448=1149.734,414.487,-89.021,-176.222,9.925,148.956
C01449=1149.730,414.734,-89.057,-176.223,9.927,148.957
C01450=1149.727,414.981,-89.094,-176.223,9.929,148.958
C01451=1149.725,415.228,-89.131,-176.224,9.931,148.958
C01452=1149.723,415.476,-89.167,-176.225,9.932,148.959
C01453=1149.722,415.698,-89.201,-176.225,9.934,148.959
C01454=1149.721,415.922,-89.234,-176.226,9.936,148.960
C01455=1149.722,416.145,-89.267,-176.226,9.937,148.961
C01456=1149.723,416.369,-89.300,-176.227,9.939,148.961
C01457=1149.723,416.591,-89.332,-176.227,9.941,148.962
C01458=1149.726,416.814,-89.365,-176.228,9.942,148.962
C01459=1149.728,417.037,-89.398,-176.228,9.944,148.963
C01460=1149.731,417.260,-89.430,-176.229,9.945,148.963
C01461=1149.312,417.261,-89.479,-176.231,9.957,148.967
C01462=1149.308,417.037,-89.447,-176.230,9.956,148.966
C01463=1149.306,416.813,-89.414,-176.230,9.954,148.966
C01464=1149.304,416.589,-89.380,-176.230,9.952,148.965
C01465=1149.302,416.364,-89.348,-176.229,9.951,148.965
C01466=1149.301,416.139,-89.314,-176.228,9.949,148.964
C01467=1149.301,415.914,-89.282,-176.228,9.947,148.964
C01468=1149.301,415.689,-89.248,-176.227,9.946,148.963
C01469=1149.303,415.464,-89.215,-176.227,9.943,148.962
C01470=1149.304,415.216,-89.178,-176.226,9.941,148.962
C01471=1149.307,414.969,-89.141,-176.226,9.940,148.961
C01472=1149.310,414.723,-89.104,-176.225,9.938,148.960
C01473=1149.314,414.475,-89.067,-176.224,9.936,148.960
C01474=1149.317,414.227,-89.030,-176.223,9.934,148.959
C01475=1149.321,413.980,-88.993,-176.223,9.932,148.958
C01476=1149.325,413.733,-88.956,-176.223,9.930,148.958
C01477=1149.329,413.486,-88.919,-176.222,9.928,148.957
C01478=1149.333,413.239,-88.883,-176.221,9.926,148.956
C01479=1149.336,412.991,-88.846,-176.220,9.924,148.955
C01480=1149.340,412.745,-88.808,-176.219,9.922,148.955
C01481=1149.344,412.497,-88.771,-176.219,9.921,148.954
C01482=1149.348,412.250,-88.735,-176.218,9.919,148.954
C01483=1149.352,412.002,-88.697,-176.217,9.917,148.953
C01484=1149.356,411.755,-88.660,-176.216,9.915,148.952
C01485=1149.359,411.508,-88.624,-176.216,9.913,148.951
C01486=1149.363,411.261,-88.587,-176.215,9.911,148.951
C01487=1149.367,411.014,-88.550,-176.214,9.909,148.950
C01488=1149.371,410.767,-88.513,-176.214,9.907,148.949
C01489=1149.375,410.519,-88.476,-176.213,9.905,148.948
C01490=1149.379,410.272,-88.439,-176.212,9.903,148.948
C01491=1149.383,410.025,-88.402,-176.211,9.901,148.947
C01492=1149.387,409.778,-88.365,-176.210,9.899,148.946
C01493=1149.390,409.530,-88.328,-176.210,9.898,148.946
C01494=1149.394,409.283,-88.292,-176.209,9.896,148.945
C01495=1149.398,409.036,-88.255,-176.208,9.894,148.944
C01496=1149.402,408.789,-88.217,-176.207,9.892,148.944
C01497=1149.405,408.541,-88.180,-176.205,9.891,148.943
C01498=1149.409,408.294,-88.143,-176.205,9.889,148.942
C01499=1149.413,408.047,-88.107,-176.204,9.887,148.941
C01500=1149.417,407.800,-88.070,-176.203,9.885,148.941
C01501=1149.421,407.553,-88.033,-176.202,9.883,148.940
C01502=1149.424,407.305,-87.996,-176.201,9.881,148.939
C01503=1149.428,407.058,-87.959,-176.201,9.880,148.939
C01504=1149.432,406.811,-87.922,-176.199,9.878,148.938
C01505=1149.436,406.564,-87.885,-176.198,9.875,148.937
C01506=1149.439,406.316,-87.848,-176.198,9.874,148.936
C01507=1149.443,406.069,-87.811,-176.197,9.872,148.935
C01508=1149.447,405.822,-87.774,-176.196,9.870,148.935
C01509=1149.451,405.575,-87.737,-176.195,9.868,148.934
C01510=1149.455,405.328,-87.701,-176.194,9.866,148.933
C01511=1149.459,405.080,-87.663,-176.193,9.864,148.932
C01512=1149.463,404.833,-87.626,-176.192,9.863,148.932
C01513=1149.466,404.586,-87.590,-176.191,9.861,148.931
C01514=1149.470,404.339,-87.553,-176.190,9.859,148.930
C01515=1149.474,404.091,-87.515,-176.189,9.857,148.930
C01516=1149.478,403.844,-87.479,-176.188,9.855,148.929
C01517=1149.482,403.597,-87.442,-176.187,9.853,148.928
C01518=1149.486,403.350,-87.405,-176.186,9.851,148.927
C01519=1149.489,403.103,-87.369,-176.185,9.849,148.926
C01520=1149.493,402.855,-87.331,-176.184,9.847,148.926
C01521=1149.497,402.608,-87.295,-176.183,9.845,148.925
C01522=1149.501,402.361,-87.258,-176.182,9.843,148.924
C01523=1149.505,402.113,-87.221,-176.180,9.842,148.923
C01524=1149.509,401.867,-87.183,-176.179,9.840,148.922
C01525=1149.512,401.619,-87.146,-176.179,9.838,148.922
C01526=1149.516,401.372,-87.110,-176.177,9.836,148.921
C01527=1149.520,401.125,-87.073,-176.176,9.834,148.920
C01528=1149.524,400.878,-87.036,-176.175,9.832,148.919
C01529=1149.527,400.630,-86.999,-176.174,9.830,148.918
C01530=1149.531,400.383,-86.962,-176.173,9.828,148.918
C01531=1149.536,400.135,-86.925,-176.172,9.826,148.917
C01532=1149.539,399.888,-86.889,-176.171,9.824,148.916
C01533=1149.543,399.642,-86.851,-176.170,9.822,148.915
C01534=1149.546,399.394,-86.814,-176.169,9.820,148.914
C01535=1149.550,399.147,-86.777,-176.168,9.818,148.914
C01536=1149.554,398.900,-86.740,-176.167,9.816,148.913
C01537=1149.558,398.652,-86.703,-176.166,9.814,148.912
C01538=1149.563,398.405,-86.667,-176.165,9.812,148.911
C01539=1149.565,398.158,-86.630,-176.164,9.810,148.910
C01540=1149.569,397.910,-86.593,-176.163,9.808,148.910
C01541=1149.574,397.663,-86.556,-176.162,9.806,148.909
C01542=1149.578,397.416,-86.519,-176.161,9.804,148.908
C01543=1149.581,397.168,-86.482,-176.160,9.801,148.907
C01544=1149.585,396.922,-86.445,-176.159,9.799,148.906
C01545=1149.588,396.675,-86.408,-176.158,9.797,148.906
C01546=1149.592,396.428,-86.371,-176.157,9.795,148.905
C01547=1149.596,396.180,-86.335,-176.156,9.793,148.904
C01548=1149.600,395.932,-86.297,-176.155,9.791,148.903
C01549=1149.604,395.685,-86.261,-176.154,9.788,148.902
C01550=1149.608,395.438,-86.224,-176.153,9.786,148.901
C01551=1149.611,395.191,-86.187,-176.152,9.784,148.900
C01552=1149.616,394.944,-86.151,-176.151,9.782,148.900
C01553=1149.619,394.696,-86.113,-176.151,9.779,148.899
C01554=1149.623,394.449,-86.076,-176.150,9.777,148.898
C01555=1149.627,394.202,-86.039,-176.149,9.775,148.897
C01556=1149.631,393.955,-86.002,-176.148,9.772,148.896
C01557=1149.634,393.708,-85.966,-176.147,9.770,148.896
C01558=1149.638,393.460,-85.929,-176.147,9.768,148.895
C01559=1149.642,393.213,-85.892,-176.146,9.765,148.894
C01560=1149.646,392.966,-85.855,-176.145,9.763,148.893
C01561=1149.650,392.719,-85.818,-176.144,9.761,148.892
C01562=1149.654,392.472,-85.781,-176.143,9.758,148.891
C01563=1149.657,392.224,-85.744,-176.143,9.756,148.891
C01564=1149.661,391.977,-85.708,-176.142,9.753,148.890
C01565=1149.665,391.730,-85.671,-176.142,9.750,148.889
C01566=1149.669,391.444,-85.628,-176.141,9.747,148.888
C01567=1149.674,391.157,-85.585,-176.140,9.744,148.887
C01568=1149.678,390.870,-85.543,-176.140,9.741,148.886
C01569=1149.683,390.584,-85.499,-176.139,9.738,148.885
C01570=1149.686,390.337,-85.463,-176.139,9.736,148.884
C01571=1149.690,390.090,-85.426,-176.137,9.733,148.883
C01572=1149.694,389.842,-85.389,-176.137,9.731,148.882
C01573=1149.698,389.594,-85.352,-176.136,9.728,148.881
C01574=1149.701,389.348,-85.316,-176.136,9.725,148.881
C01575=1149.705,389.100,-85.279,-176.136,9.722,148.880
C01576=1149.710,388.853,-85.242,-176.136,9.719,148.879
C01577=1149.713,388.605,-85.205,-176.136,9.716,148.878
C01578=1149.717,388.358,-85.168,-176.135,9.713,148.877
C01579=1149.720,388.111,-85.132,-176.135,9.711,148.877
C01580=1149.725,387.864,-85.095,-176.135,9.708,148.876
C01581=1149.729,387.617,-85.058,-176.135,9.704,148.875
C01582=1149.732,387.369,-85.021,-176.134,9.701,148.874
C01583=1149.736,387.122,-84.985,-176.135,9.698,148.873
C01584=1149.740,386.875,-84.948,-176.134,9.695,148.872
C01585=1149.744,386.628,-84.911,-176.135,9.692,148.872
C01586=1149.748,386.380,-84.874,-176.134,9.689,148.871
C01587=1149.752,386.133,-84.837,-176.135,9.686,148.870
C01588=1149.755,385.886,-84.800,-176.135,9.682,148.869
C01589=1149.759,385.639,-84.764,-176.135,9.680,148.869
C01590=1149.763,385.391,-84.727,-176.135,9.676,148.868
C01591=1149.766,385.144,-84.691,-176.136,9.673,148.867
C01592=1149.770,384.897,-84.654,-176.136,9.669,148.866
C01593=1149.774,384.650,-84.617,-176.137,9.666,148.865
C01594=1149.778,384.402,-84.580,-176.137,9.662,148.865
C01595=1149.781,384.155,-84.543,-176.138,9.659,148.864
C01596=1149.786,383.907,-84.507,-176.138,9.656,148.863
C01597=1149.790,383.660,-84.470,-176.139,9.651,148.862
C01598=1149.794,383.413,-84.433,-176.140,9.648,148.862
C01599=1149.797,383.166,-84.397,-176.141,9.645,148.861
C01600=1149.801,382.919,-84.360,-176.142,9.641,148.860
C01601=1149.805,382.671,-84.323,-176.142,9.637,148.859
C01602=1149.808,382.424,-84.287,-176.144,9.634,148.859
C01603=1149.813,382.176,-84.251,-176.144,9.630,148.858
C01604=1149.817,381.929,-84.214,-176.145,9.626,148.857
C01605=1149.820,381.682,-84.178,-176.147,9.622,148.856
C01606=1149.824,381.435,-84.141,-176.147,9.619,148.856
C01607=1149.828,381.188,-84.104,-176.149,9.615,148.855
C01608=1149.832,380.941,-84.068,-176.150,9.611,148.854
C01609=1149.836,380.693,-84.031,-176.151,9.607,148.854
C01610=1149.839,380.445,-83.994,-176.153,9.603,148.853
C01611=1149.843,380.199,-83.958,-176.154,9.599,148.852
C01612=1149.847,379.951,-83.921,-176.155,9.595,148.852
C01613=1149.851,379.704,-83.886,-176.157,9.591,148.851
C01614=1149.855,379.457,-83.849,-176.158,9.587,148.851
C01615=1149.859,379.209,-83.812,-176.160,9.583,148.850
C01616=1149.862,378.962,-83.776,-176.161,9.579,148.849
C01617=1149.866,378.715,-83.739,-176.163,9.576,148.849
C01618=1149.870,378.468,-83.703,-176.164,9.572,148.848
C01619=1149.874,378.220,-83.667,-176.166,9.568,148.848
C01620=1149.878,377.973,-83.630,-176.168,9.563,148.847
C01621=1149.882,377.726,-83.594,-176.170,9.560,148.846
C01622=1149.886,377.478,-83.558,-176.171,9.556,148.846
C01623=1149.889,377.231,-83.522,-176.173,9.551,148.845
C01624=1149.894,376.984,-83.485,-176.175,9.547,148.845
C01625=1149.897,376.737,-83.449,-176.177,9.543,148.844
C01626=1149.901,376.489,-83.412,-176.179,9.539,148.844
C01627=1149.905,376.242,-83.377,-176.181,9.535,148.843
C01628=1149.909,375.995,-83.340,-176.183,9.531,148.843
C01629=1149.913,375.747,-83.304,-176.185,9.527,148.842
C01630=1149.917,375.500,-83.267,-176.187,9.523,148.841
C01631=1149.920,375.253,-83.232,-176.189,9.519,148.841
C01632=1149.925,375.005,-83.195,-176.191,9.514,148.840
C01633=1149.928,374.758,-83.159,-176.193,9.511,148.840
C01634=1149.932,374.511,-83.123,-176.195,9.506,148.839
C01635=1149.936,374.263,-83.087,-176.197,9.502,148.839
C01636=1149.940,374.016,-83.052,-176.199,9.498,148.838
C01637=1149.944,373.768,-83.015,-176.201,9.494,148.838
C01638=1149.947,373.521,-82.979,-176.204,9.490,148.837
C01639=1149.952,373.274,-82.942,-176.206,9.486,148.837
C01640=1149.955,373.026,-82.907,-176.208,9.482,148.837
C01641=1149.959,372.779,-82.871,-176.211,9.478,148.836
C01642=1149.963,372.532,-82.834,-176.213,9.473,148.836
C01643=1149.967,372.284,-82.799,-176.215,9.470,148.835
C01644=1149.971,372.036,-82.763,-176.218,9.465,148.835
C01645=1149.974,371.789,-82.726,-176.220,9.461,148.834
C01646=1149.978,371.542,-82.691,-176.222,9.457,148.834
C01647=1149.982,371.294,-82.655,-176.224,9.453,148.833
C01648=1149.986,371.047,-82.619,-176.227,9.448,148.833
C01649=1149.989,370.800,-82.583,-176.229,9.444,148.832
C01650=1149.994,370.552,-82.547,-176.232,9.441,148.832
C01651=1149.998,370.305,-82.512,-176.234,9.436,148.832
C01652=1150.002,370.058,-82.476,-176.237,9.432,148.831
C01653=1150.005,369.810,-82.440,-176.239,9.428,148.831
C01654=1150.010,369.563,-82.404,-176.242,9.424,148.831
C01655=1150.013,369.315,-82.368,-176.244,9.420,148.830
C01656=1150.017,369.068,-82.332,-176.246,9.416,148.830
C01657=1150.021,368.820,-82.297,-176.249,9.411,148.829
C01658=1150.026,368.573,-82.261,-176.251,9.408,148.829
C01659=1150.029,368.326,-82.226,-176.254,9.403,148.829
C01660=1150.033,368.078,-82.190,-176.257,9.399,148.828
C01661=1150.036,367.831,-82.155,-176.259,9.395,148.828
C01662=1150.040,367.583,-82.119,-176.262,9.392,148.828
C01663=1150.045,367.335,-82.083,-176.264,9.387,148.827
C01664=1150.049,367.089,-82.048,-176.266,9.383,148.827
C01665=1150.052,366.841,-82.012,-176.269,9.379,148.826
C01666=1150.056,366.594,-81.977,-176.271,9.375,148.826
C01667=1150.060,366.346,-81.941,-176.274,9.371,148.826
C01668=1150.064,366.098,-81.905,-176.277,9.367,148.825
C01669=1150.068,365.852,-81.870,-176.280,9.363,148.825
C01670=1150.073,365.568,-81.829,-176.282,9.358,148.824
C01671=1150.077,365.285,-81.789,-176.286,9.353,148.824
C01672=1150.081,365.002,-81.748,-176.288,9.349,148.824
C01673=1150.085,364.718,-81.707,-176.292,9.344,148.823
C01674=1150.090,364.472,-81.672,-176.293,9.340,148.823
C01675=1150.093,364.224,-81.636,-176.296,9.336,148.823
C01676=1150.097,363.976,-81.602,-176.299,9.332,148.822
C01677=1150.101,363.728,-81.566,-176.302,9.328,148.822
C01678=1150.105,363.482,-81.531,-176.304,9.325,148.822
C01679=1150.109,363.234,-81.495,-176.307,9.320,148.821
C01680=1150.113,362.987,-81.460,-176.309,9.316,148.821
C01681=1150.117,362.739,-81.425,-176.311,9.313,148.821
C01682=1150.121,362.492,-81.390,-176.314,9.308,148.820
C01683=1150.124,362.244,-81.354,-176.317,9.304,148.820
C01684=1150.128,361.996,-81.319,-176.320,9.300,148.820
C01685=1150.133,361.749,-81.284,-176.322,9.297,148.819
C01686=1150.136,361.502,-81.249,-176.324,9.292,148.819
C01687=1150.140,361.254,-81.214,-176.327,9.288,148.819
C01688=1150.144,361.006,-81.178,-176.330,9.285,148.818
C01689=1150.148,360.759,-81.143,-176.332,9.281,148.818
C01690=1150.152,360.511,-81.108,-176.335,9.276,148.818
C01691=1150.156,360.264,-81.073,-176.337,9.273,148.817
C01692=1150.160,360.016,-81.038,-176.340,9.269,148.817
C01693=1150.164,359.769,-81.003,-176.343,9.265,148.817
C01694=1150.167,359.521,-80.968,-176.345,9.261,148.816
C01695=1150.172,359.274,-80.933,-176.348,9.257,148.816
C01696=1150.175,359.027,-80.898,-176.350,9.253,148.816
C01697=1150.180,358.779,-80.863,-176.352,9.249,148.815
C01698=1150.183,358.532,-80.828,-176.355,9.245,148.815
C01699=1150.187,358.284,-80.793,-176.358,9.241,148.815
C01700=1150.192,358.036,-80.758,-176.360,9.238,148.814
C01701=1150.195,357.789,-80.723,-176.363,9.234,148.814
C01702=1150.199,357.541,-80.689,-176.366,9.229,148.814
C01703=1150.203,357.294,-80.653,-176.368,9.226,148.813
C01704=1150.207,357.046,-80.619,-176.370,9.221,148.813
C01705=1150.212,356.799,-80.584,-176.373,9.218,148.813
C01706=1150.215,356.551,-80.549,-176.376,9.214,148.813
C01707=1150.219,356.303,-80.514,-176.378,9.210,148.812
C01708=1150.223,356.057,-80.479,-176.380,9.206,148.812
C01709=1150.227,355.808,-80.444,-176.383,9.202,148.811
C01710=1150.231,355.561,-80.410,-176.385,9.199,148.811
C01711=1150.235,355.313,-80.376,-176.388,9.195,148.811
C01712=1150.239,355.066,-80.340,-176.390,9.191,148.811
C01713=1150.243,354.818,-80.306,-176.393,9.187,148.810
C01714=1150.247,354.571,-80.272,-176.396,9.183,148.810
C01715=1150.251,354.323,-80.237,-176.398,9.179,148.810
C01716=1150.255,354.076,-80.202,-176.401,9.175,148.809
C01717=1150.258,353.828,-80.167,-176.403,9.172,148.809
C01718=1150.262,353.580,-80.133,-176.405,9.168,148.809
C01719=1150.267,353.333,-80.098,-176.408,9.164,148.808
C01720=1150.270,353.085,-80.064,-176.411,9.160,148.808
C01721=1150.275,352.838,-80.029,-176.413,9.156,148.808
C01722=1150.278,352.590,-79.994,-176.415,9.152,148.808
C01723=1150.282,352.343,-79.960,-176.418,9.148,148.807
C01724=1150.287,352.096,-79.926,-176.420,9.145,148.807
C01725=1150.291,351.848,-79.891,-176.423,9.141,148.807
C01726=1150.294,351.600,-79.857,-176.425,9.137,148.806
C01727=1150.298,351.352,-79.822,-176.428,9.133,148.806
C01728=1150.302,351.105,-79.788,-176.430,9.130,148.806
C01729=1150.306,350.857,-79.753,-176.433,9.126,148.805
C01730=1150.311,350.610,-79.719,-176.436,9.121,148.805
C01731=1150.314,350.362,-79.685,-176.438,9.118,148.805
C01732=1150.319,350.114,-79.650,-176.441,9.114,148.805
C01733=1150.322,349.867,-79.616,-176.443,9.110,148.804
C01734=1150.326,349.619,-79.581,-176.446,9.106,148.804
C01735=1150.330,349.372,-79.548,-176.448,9.103,148.804
C01736=1150.334,349.124,-79.513,-176.451,9.099,148.803
C01737=1150.338,348.877,-79.479,-176.453,9.095,148.803
C01738=1150.342,348.629,-79.444,-176.456,9.091,148.803
C01739=1150.346,348.381,-79.411,-176.458,9.088,148.803
C01740=1150.351,348.134,-79.376,-176.460,9.084,148.802
C01741=1150.354,347.886,-79.342,-176.463,9.080,148.802
C01742=1150.358,347.638,-79.308,-176.466,9.076,148.802
C01743=1150.362,347.391,-79.274,-176.469,9.072,148.801
C01744=1150.366,347.143,-79.239,-176.471,9.069,148.801
C01745=1150.370,346.895,-79.206,-176.473,9.064,148.801
C01746=1150.374,346.647,-79.171,-176.476,9.061,148.801
C01747=1150.378,346.400,-79.137,-176.479,9.057,148.800
C01748=1150.382,346.153,-79.103,-176.481,9.053,148.800
C01749=1150.386,345.904,-79.069,-176.483,9.049,148.800
C01750=1150.390,345.657,-79.035,-176.486,9.046,148.799
C01751=1150.395,345.410,-79.001,-176.489,9.042,148.799
C01752=1150.398,345.161,-78.967,-176.491,9.038,148.799
C01753=1150.402,344.914,-78.933,-176.493,9.034,148.798
C01754=1150.407,344.667,-78.899,-176.496,9.031,148.798
C01755=1150.411,344.419,-78.866,-176.499,9.027,148.798
C01756=1150.414,344.171,-78.832,-176.501,9.024,148.798
C01757=1150.419,343.924,-78.797,-176.503,9.019,148.797
C01758=1150.423,343.676,-78.764,-176.506,9.016,148.797
C01759=1150.426,343.428,-78.730,-176.509,9.012,148.797
C01760=1150.431,343.180,-78.696,-176.511,9.009,148.797
C01761=1150.435,342.933,-78.662,-176.514,9.005,148.796
C01762=1150.439,342.685,-78.629,-176.516,9.001,148.796
C01763=1150.443,342.437,-78.594,-176.519,8.997,148.796
C01764=1150.447,342.190,-78.561,-176.521,8.994,148.796
C01765=1150.451,341.942,-78.527,-176.524,8.990,148.795
C01766=1150.455,341.695,-78.494,-176.526,8.986,148.795
C01767=1150.459,341.447,-78.459,-176.529,8.982,148.795
C01768=1150.463,341.199,-78.426,-176.531,8.979,148.795
C01769=1150.467,340.952,-78.392,-176.534,8.975,148.794
C01770=1150.471,340.704,-78.359,-176.536,8.971,148.794
C01771=1150.475,340.456,-78.324,-176.539,8.967,148.794
C01772=1150.479,340.208,-78.291,-176.542,8.964,148.794
C01773=1150.483,339.960,-78.258,-176.543,8.960,148.793
C01774=1150.488,339.680,-78.219,-176.547,8.955,148.793
C01775=1150.493,339.400,-78.182,-176.550,8.951,148.793
C01776=1150.497,339.120,-78.144,-176.553,8.947,148.792
C01777=1150.502,338.840,-78.106,-176.556,8.943,148.792
C01778=1150.506,338.592,-78.073,-176.558,8.940,148.792
C01779=1150.509,338.345,-78.038,-176.560,8.935,148.792
C01780=1150.513,338.097,-78.005,-176.563,8.932,148.791
C01781=1150.518,337.849,-77.972,-176.566,8.928,148.791
C01782=1150.521,337.602,-77.938,-176.568,8.925,148.791
C01783=1150.525,337.354,-77.905,-176.570,8.922,148.791
C01784=1150.530,337.107,-77.872,-176.573,8.917,148.790
C01785=1150.534,336.858,-77.838,-176.576,8.914,148.790
C01786=1150.538,336.610,-77.805,-176.578,8.910,148.790
C01787=1150.542,336.363,-77.771,-176.581,8.907,148.790
C01788=1150.546,336.115,-77.738,-176.583,8.902,148.789
C01789=1150.550,335.867,-77.704,-176.586,8.899,148.789
C01790=1150.554,335.620,-77.671,-176.588,8.895,148.789
C01791=1150.558,335.372,-77.638,-176.591,8.892,148.789
C01792=1150.563,335.124,-77.605,-176.593,8.888,148.788
C01793=1150.566,334.876,-77.571,-176.596,8.884,148.788
C01794=1150.570,334.628,-77.538,-176.598,8.881,148.788
C01795=1150.574,334.380,-77.505,-176.601,8.877,148.788
C01796=1150.578,334.133,-77.472,-176.604,8.874,148.788
C01797=1150.583,333.885,-77.439,-176.606,8.870,148.787
C01798=1150.587,333.637,-77.406,-176.609,8.866,148.787
C01799=1150.591,333.389,-77.372,-176.611,8.863,148.787
C01800=1150.595,333.142,-77.339,-176.614,8.859,148.787
C01801=1150.598,332.894,-77.307,-176.616,8.855,148.786
C01802=1150.603,332.647,-77.274,-176.619,8.851,148.786
C01803=1150.607,332.399,-77.240,-176.621,8.848,148.786
C01804=1150.611,332.151,-77.207,-176.624,8.844,148.786
C01805=1150.615,331.903,-77.174,-176.626,8.841,148.785
C01806=1150.619,331.656,-77.141,-176.629,8.837,148.785
C01807=1150.623,331.408,-77.108,-176.632,8.833,148.785
C01808=1150.627,331.160,-77.075,-176.634,8.830,148.785
C01809=1150.632,330.913,-77.042,-176.637,8.826,148.785
C01810=1150.635,330.664,-77.010,-176.639,8.823,148.784
C01811=1150.639,330.417,-76.977,-176.641,8.819,148.784
C01812=1150.644,330.169,-76.943,-176.644,8.815,148.784
